LIN {X 0,Y 425.307,Z 310.007,A -85,B 0,C 180,E1 -9738.298,E2 -9738.298} C_VEL
LIN {X 0,Y 425.293,Z 310.002,A -85,B 0,C 180,E1 -9741.318,E2 -9741.318} C_VEL
LIN {X 0,Y 425.3,Z 309.999,A -85,B 0,C 180,E1 -9744.651,E2 -9744.651} C_VEL
LIN {X 0,Y 425.25,Z 310.01,A -85,B 0,C 180,E1 -9747.564,E2 -9747.564} C_VEL
LIN {X 0,Y 425.28,Z 310.001,A -85,B 0,C 180,E1 -9749.72,E2 -9749.72} C_VEL
LIN {X 0,Y 425.269,Z 310.007,A -85,B 0,C 180,E1 -9753.049,E2 -9753.049} C_VEL
LIN {X 0,Y 425.279,Z 310.005,A -85,B 0,C 180,E1 -9755.928,E2 -9755.928} C_VEL
LIN {X 0,Y 425.258,Z 310.007,A -85,B 0,C 180,E1 -9759.036,E2 -9759.036} C_VEL
LIN {X 0,Y 425.253,Z 310.008,A -85,B 0,C 180,E1 -9762.655,E2 -9762.655} C_VEL
LIN {X 0,Y 425.281,Z 310.005,A -85,B 0,C 180,E1 -9765.283,E2 -9765.283} C_VEL
LIN {X 0,Y 425.245,Z 310.016,A -85,B 0,C 180,E1 -9768.618,E2 -9768.618} C_VEL
LIN {X 0,Y 425.277,Z 310.011,A -85,B 0,C 180,E1 -9771.099,E2 -9771.099} C_VEL
LIN {X 0,Y 425.293,Z 310.007,A -85,B 0,C 180,E1 -9774.663,E2 -9774.663} C_VEL
LIN {X 0,Y 425.261,Z 310.012,A -85,B 0,C 180,E1 -9778.073,E2 -9778.073} C_VEL
LIN {X 0,Y 425.311,Z 310.005,A -85,B 0,C 180,E1 -9781.366,E2 -9781.366} C_VEL
LIN {X 0,Y 425.335,Z 310.116,A -85,B 0,C 180,E1 -9783.702,E2 -9783.702} C_VEL
LIN {X 0,Y 427.72,Z 322.373,A -85,B 0,C 180,E1 -9786.518,E2 -9786.518} C_VEL
LIN {X 0,Y 427.919,Z 326.115,A -85,B 0,C 180,E1 -9787.322,E2 -9787.322} C_VEL
LIN {X 0,Y 426.781,Z 342.849,A -85,B 0,C 180,E1 -9790.771,E2 -9790.771} C_VEL
LIN {X 0,Y 426.66,Z 345.828,A -85,B 0,C 180,E1 -9791.314,E2 -9791.314} C_VEL
LIN {X 0,Y 430.359,Z 367.602,A -85,B 0,C 180,E1 -9791.874,E2 -9791.874} C_VEL
LIN {X 0,Y 429.563,Z 451.981,A -85,B 0,C 180,E1 -9793.332,E2 -9793.332} C_VEL
LIN {X 0,Y 429.279,Z 461.728,A -85,B 0,C 180,E1 -9793.596,E2 -9793.596} C_VEL
LIN {X 0,Y 428.817,Z 472.261,A -85,B 0,C 180,E1 -9794.005,E2 -9794.005} C_VEL
LIN {X 0,Y 428.352,Z 482.441,A -85,B 0,C 180,E1 -9794.537,E2 -9794.537} C_VEL
LIN {X 0,Y 427.723,Z 493.013,A -85,B 0,C 180,E1 -9795.245,E2 -9795.245} C_VEL
LIN {X 0,Y 427.159,Z 502.459,A -85,B 0,C 180,E1 -9796.031,E2 -9796.031} C_VEL
LIN {X 0,Y 426.599,Z 511.193,A -85,B 0,C 180,E1 -9796.907,E2 -9796.907} C_VEL
LIN {X 0,Y 426.058,Z 519.156,A -85,B 0,C 180,E1 -9797.859,E2 -9797.859} C_VEL
LIN {X 0,Y 425.479,Z 527.402,A -85,B 0,C 180,E1 -9799.05,E2 -9799.05} C_VEL
LIN {X 0,Y 425.032,Z 534.27,A -85,B 0,C 180,E1 -9800.242,E2 -9800.242} C_VEL
LIN {X 0,Y 424.705,Z 540.013,A -85,B 0,C 180,E1 -9801.435,E2 -9801.435} C_VEL
LIN {X 0,Y 424.433,Z 545.574,A -85,B 0,C 180,E1 -9802.866,E2 -9802.866} C_VEL
LIN {X 0,Y 424.231,Z 549.948,A -85,B 0,C 180,E1 -9804.295,E2 -9804.295} C_VEL
LIN {X 0,Y 424.204,Z 552.264,A -85,B 0,C 180,E1 -9805.248,E2 -9805.248} C_VEL
LIN {X 0,Y 424.081,Z 555.578,A -85,B 0,C 180,E1 -9807.15,E2 -9807.15} C_VEL
LIN {X 0,Y 424.115,Z 556.545,A -85,B 0,C 180,E1 -9808.101,E2 -9808.101} C_VEL
LIN {X 0,Y 424.056,Z 557.441,A -85,B 0,C 180,E1 -9810,E2 -9810} C_VEL
LIN {X 0,Y 424.115,Z 556.603,A -85,B 0,C 180,E1 -9811.899,E2 -9811.899} C_VEL
LIN {X 0,Y 424.081,Z 555.632,A -85,B 0,C 180,E1 -9812.85,E2 -9812.85} C_VEL
LIN {X 0,Y 424.209,Z 552.407,A -85,B 0,C 180,E1 -9814.752,E2 -9814.752} C_VEL
LIN {X 0,Y 424.262,Z 548.344,A -85,B 0,C 180,E1 -9816.328,E2 -9816.328} C_VEL
LIN {X 0,Y 424.502,Z 544.103,A -85,B 0,C 180,E1 -9817.611,E2 -9817.611} C_VEL
LIN {X 0,Y 424.848,Z 538.126,A -85,B 0,C 180,E1 -9819.042,E2 -9819.042} C_VEL
LIN {X 0,Y 425.237,Z 532.082,A -85,B 0,C 180,E1 -9820.234,E2 -9820.234} C_VEL
LIN {X 0,Y 425.716,Z 524.793,A -85,B 0,C 180,E1 -9821.426,E2 -9821.426} C_VEL
LIN {X 0,Y 426.395,Z 515.929,A -85,B 0,C 180,E1 -9822.614,E2 -9822.614} C_VEL
LIN {X 0,Y 426.936,Z 506.91,A -85,B 0,C 180,E1 -9823.618,E2 -9823.618} C_VEL
LIN {X 0,Y 427.6,Z 497.037,A -85,B 0,C 180,E1 -9824.516,E2 -9824.516} C_VEL
LIN {X 0,Y 428.15,Z 487.502,A -85,B 0,C 180,E1 -9825.227,E2 -9825.227} C_VEL
LIN {X 0,Y 428.764,Z 477.643,A -85,B 0,C 180,E1 -9825.813,E2 -9825.813} C_VEL
LIN {X 0,Y 429.288,Z 465.878,A -85,B 0,C 180,E1 -9826.343,E2 -9826.343} C_VEL
LIN {X 0,Y 429.644,Z 455.964,A -85,B 0,C 180,E1 -9826.665,E2 -9826.665} C_VEL
LIN {X 0,Y 429.921,Z 439.713,A -85,B 0,C 180,E1 -9826.99,E2 -9826.99} C_VEL
LIN {X 0,Y 430.624,Z 368.061,A -85,B 0,C 180,E1 -9828.215,E2 -9828.215} C_VEL
LIN {X 0,Y 426.817,Z 345.669,A -85,B 0,C 180,E1 -9828.806,E2 -9828.806} C_VEL
LIN {X 0,Y 426.763,Z 344.428,A -85,B 0,C 180,E1 -9828.969,E2 -9828.969} C_VEL
LIN {X 0,Y 427.787,Z 327.218,A -85,B 0,C 180,E1 -9832.439,E2 -9832.439} C_VEL
LIN {X 0,Y 427.876,Z 323.444,A -85,B 0,C 180,E1 -9833.216,E2 -9833.216} C_VEL
LIN {X 0,Y 425.789,Z 312.361,A -85,B 0,C 180,E1 -9835.676,E2 -9835.676} C_VEL
LIN {X 0,Y 425.31,Z 310.053,A -85,B 0,C 180,E1 -9836.266,E2 -9836.266} C_VEL
LIN {X 0,Y 425.283,Z 310.01,A -85,B 0,C 180,E1 -9839.72,E2 -9839.72} C_VEL
LIN {X 0,Y 425.279,Z 310.009,A -85,B 0,C 180,E1 -9843.048,E2 -9843.048} C_VEL
LIN {X 0,Y 425.279,Z 310.009,A -85,B 0,C 180,E1 -9845.929,E2 -9845.929} C_VEL
LIN {X 0,Y 425.28,Z 310.008,A -85,B 0,C 180,E1 -9849.041,E2 -9849.041} C_VEL
LIN {X 0,Y 425.28,Z 310.007,A -85,B 0,C 180,E1 -9851.957,E2 -9851.957} C_VEL
LIN {X 0,Y 425.283,Z 310.011,A -85,B 0,C 180,E1 -9855.283,E2 -9855.283} C_VEL
LIN {X 0,Y 425.272,Z 310.004,A -85,B 0,C 180,E1 -9858.622,E2 -9858.622} C_VEL
LIN {X 0,Y 425.296,Z 310.005,A -85,B 0,C 180,E1 -9861.101,E2 -9861.101} C_VEL
LIN {X 0,Y 425.299,Z 310.001,A -85,B 0,C 180,E1 -9864.664,E2 -9864.664} C_VEL
LIN {X 0,Y 425.265,Z 310.012,A -85,B 0,C 180,E1 -9868.073,E2 -9868.073} C_VEL
LIN {X 0,Y 425.331,Z 309.999,A -85,B 0,C 180,E1 -9871.368,E2 -9871.368} C_VEL
LIN {X 0,Y 425.296,Z 310.009,A -85,B 0,C 180,E1 -9874.555,E2 -9874.555} C_VEL
LIN {X 0,Y 425.288,Z 310.004,A -85,B 0,C 180,E1 -9877.662,E2 -9877.662} C_VEL
LIN {X 0,Y 425.363,Z 309.997,A -85,B 0,C 180,E1 -9880.704,E2 -9880.704} C_VEL
LIN {X 0,Y 425.389,Z 309.996,A -85,B 0,C 180,E1 -9883.689,E2 -9883.689} C_VEL
LIN {X 0,Y 425.413,Z 309.991,A -85,B 0,C 180,E1 -9887.599,E2 -9887.599} C_VEL
LIN {X 0,Y 425.444,Z 309.981,A -85,B 0,C 180,E1 -9891.45,E2 -9891.45} C_VEL
LIN {X 0,Y 425.556,Z 309.974,A -85,B 0,C 180,E1 -9894.314,E2 -9894.314} C_VEL
LIN {X 0,Y 425.577,Z 309.972,A -85,B 0,C 180,E1 -9898.108,E2 -9898.108} C_VEL
LIN {X 0,Y 425.705,Z 309.952,A -85,B 0,C 180,E1 -9900,E2 -9900} C_VEL
LIN {X 0,Y 425.558,Z 309.978,A -85,B 0,C 180,E1 -9902.84,E2 -9902.84} C_VEL
LIN {X 0,Y 425.534,Z 309.977,A -85,B 0,C 180,E1 -9906.639,E2 -9906.639} C_VEL
LIN {X 0,Y 425.403,Z 309.995,A -85,B 0,C 180,E1 -9909.51,E2 -9909.51} C_VEL
LIN {X 0,Y 425.395,Z 309.989,A -85,B 0,C 180,E1 -9912.904,E2 -9912.904} C_VEL
LIN {X 0,Y 425.363,Z 309.995,A -85,B 0,C 180,E1 -9916.605,E2 -9916.605} C_VEL
LIN {X 0,Y 425.33,Z 310.001,A -85,B 0,C 180,E1 -9919.636,E2 -9919.636} C_VEL
LIN {X 0,Y 425.289,Z 310.01,A -85,B 0,C 180,E1 -9922.339,E2 -9922.339} C_VEL
LIN {X 0,Y 425.321,Z 310.006,A -85,B 0,C 180,E1 -9924.657,E2 -9924.657} C_VEL
LIN {X 0,Y 425.33,Z 309.992,A -85,B 0,C 180,E1 -9927.559,E2 -9927.559} C_VEL
LIN {X 0,Y 425.288,Z 310.006,A -85,B 0,C 180,E1 -9930.816,E2 -9930.816} C_VEL
LIN {X 0,Y 425.31,Z 310,A -85,B 0,C 180,E1 -9934.288,E2 -9934.288} C_VEL
LIN {X 0,Y 425.28,Z 310.01,A -85,B 0,C 180,E1 -9937.694,E2 -9937.694} C_VEL
LIN {X 0,Y 425.282,Z 310.011,A -85,B 0,C 180,E1 -9940.521,E2 -9940.521} C_VEL
LIN {X 0,Y 425.357,Z 310.083,A -85,B 0,C 180,E1 -9942.153,E2 -9942.153} C_VEL
LIN {X 0,Y 427.263,Z 319.771,A -85,B 0,C 180,E1 -9944.345,E2 -9944.345} C_VEL
LIN {X 0,Y 427.059,Z 329.794,A -85,B 0,C 180,E1 -9946.394,E2 -9946.394} C_VEL
LIN {X 0,Y 426.921,Z 334.032,A -85,B 0,C 180,E1 -9947.212,E2 -9947.212} C_VEL
LIN {X 0,Y 429.955,Z 350.192,A -85,B 0,C 180,E1 -9947.681,E2 -9947.681} C_VEL
LIN {X 0,Y 430.785,Z 356.193,A -85,B 0,C 180,E1 -9947.827,E2 -9947.827} C_VEL
LIN {X 0,Y 429.735,Z 440.182,A -85,B 0,C 180,E1 -9949.279,E2 -9949.279} C_VEL
LIN {X 0,Y 429.469,Z 450.36,A -85,B 0,C 180,E1 -9949.557,E2 -9949.557} C_VEL
LIN {X 0,Y 429.107,Z 461.311,A -85,B 0,C 180,E1 -9949.996,E2 -9949.996} C_VEL
LIN {X 0,Y 428.692,Z 470.759,A -85,B 0,C 180,E1 -9950.493,E2 -9950.493} C_VEL
LIN {X 0,Y 428.167,Z 480.146,A -85,B 0,C 180,E1 -9951.109,E2 -9951.109} C_VEL
LIN {X 0,Y 427.483,Z 490.943,A -85,B 0,C 180,E1 -9952.006,E2 -9952.006} C_VEL
LIN {X 0,Y 426.841,Z 499.891,A -85,B 0,C 180,E1 -9952.912,E2 -9952.912} C_VEL
LIN {X 0,Y 426.228,Z 508.549,A -85,B 0,C 180,E1 -9953.974,E2 -9953.974} C_VEL
LIN {X 0,Y 425.731,Z 515.487,A -85,B 0,C 180,E1 -9954.982,E2 -9954.982} C_VEL
LIN {X 0,Y 425.269,Z 521.992,A -85,B 0,C 180,E1 -9956.099,E2 -9956.099} C_VEL
LIN {X 0,Y 424.842,Z 528.755,A -85,B 0,C 180,E1 -9957.53,E2 -9957.53} C_VEL
LIN {X 0,Y 424.596,Z 532.91,A -85,B 0,C 180,E1 -9958.574,E2 -9958.574} C_VEL
LIN {X 0,Y 424.31,Z 537.98,A -85,B 0,C 180,E1 -9960.205,E2 -9960.205} C_VEL
LIN {X 0,Y 424.173,Z 540.902,A -85,B 0,C 180,E1 -9961.419,E2 -9961.419} C_VEL
LIN {X 0,Y 423.931,Z 544.018,A -85,B 0,C 180,E1 -9963.41,E2 -9963.41} C_VEL
LIN {X 0,Y 423.878,Z 545.06,A -85,B 0,C 180,E1 -9964.464,E2 -9964.464} C_VEL
LIN {X 0,Y 423.861,Z 545.528,A -85,B 0,C 180,E1 -9965.777,E2 -9965.777} C_VEL
LIN {X 0,Y 423.884,Z 545.029,A -85,B 0,C 180,E1 -9967.583,E2 -9967.583} C_VEL
LIN {X 0,Y 423.949,Z 543.998,A -85,B 0,C 180,E1 -9968.611,E2 -9968.611} C_VEL
LIN {X 0,Y 424.158,Z 540.764,A -85,B 0,C 180,E1 -9970.647,E2 -9970.647} C_VEL
LIN {X 0,Y 424.367,Z 536.989,A -85,B 0,C 180,E1 -9972.159,E2 -9972.159} C_VEL
LIN {X 0,Y 424.642,Z 531.745,A -85,B 0,C 180,E1 -9973.725,E2 -9973.725} C_VEL
LIN {X 0,Y 424.97,Z 525.693,A -85,B 0,C 180,E1 -9975.147,E2 -9975.147} C_VEL
LIN {X 0,Y 425.107,Z 523.362,A -85,B 0,C 180,E1 -9975.621,E2 -9975.621} C_VEL
LIN {X 0,Y 424.646,Z 520.061,A -85,B 0,C 180,E1 -9976.279,E2 -9976.279} C_VEL
LIN {X 0,Y 422.208,Z 514.295,A -85,B 0,C 180,E1 -9977.326,E2 -9977.326} C_VEL
LIN {X 0,Y 419.867,Z 507.939,A -85,B 0,C 180,E1 -9978.31,E2 -9978.31} C_VEL
LIN {X 0,Y 419.551,Z 503.63,A -85,B 0,C 180,E1 -9978.862,E2 -9978.862} C_VEL
LIN {X 0,Y 420.065,Z 495.684,A -85,B 0,C 180,E1 -9979.761,E2 -9979.761} C_VEL
LIN {X 0,Y 420.787,Z 486.221,A -85,B 0,C 180,E1 -9980.642,E2 -9980.642} C_VEL
LIN {X 0,Y 421.298,Z 476.851,A -85,B 0,C 180,E1 -9981.365,E2 -9981.365} C_VEL
LIN {X 0,Y 421.868,Z 465.719,A -85,B 0,C 180,E1 -9982.04,E2 -9982.04} C_VEL
LIN {X 0,Y 422.3,Z 455.141,A -85,B 0,C 180,E1 -9982.529,E2 -9982.529} C_VEL
LIN {X 0,Y 422.723,Z 443.786,A -85,B 0,C 180,E1 -9982.897,E2 -9982.897} C_VEL
LIN {X 0,Y 422.945,Z 427.148,A -85,B 0,C 180,E1 -9983.231,E2 -9983.231} C_VEL
LIN {X 0,Y 423.736,Z 355.549,A -85,B 0,C 180,E1 -9984.465,E2 -9984.465} C_VEL
LIN {X 0,Y 419.957,Z 335.166,A -85,B 0,C 180,E1 -9985.014,E2 -9985.014} C_VEL
LIN {X 0,Y 419.936,Z 333.83,A -85,B 0,C 180,E1 -9985.2,E2 -9985.2} C_VEL
LIN {X 0,Y 420.578,Z 323.19,A -85,B 0,C 180,E1 -9987.606,E2 -9987.606} C_VEL
LIN {X 0,Y 419.096,Z 313.301,A -85,B 0,C 180,E1 -9990,E2 -9990} C_VEL
LIN {X 0,Y 418.58,Z 310.893,A -85,B 0,C 180,E1 -9990.661,E2 -9990.661} C_VEL
LIN {X 0,Y 418.511,Z 310.857,A -85,B 0,C 180,E1 -9992.888,E2 -9992.888} C_VEL
LIN {X 0,Y 418.507,Z 310.849,A -85,B 0,C 180,E1 -9995.783,E2 -9995.783} C_VEL
LIN {X 0,Y 418.38,Z 310.864,A -85,B 0,C 180,E1 -9998.696,E2 -9998.696} C_VEL
LIN {X 0,Y 418.318,Z 310.873,A -85,B 0,C 180,E1 -10001.631,E2 -10001.631} C_VEL
LIN {X 0,Y 418.304,Z 310.874,A -85,B 0,C 180,E1 -10004.597,E2 -10004.597} C_VEL
LIN {X 0,Y 418.29,Z 310.88,A -85,B 0,C 180,E1 -10007.604,E2 -10007.604} C_VEL
LIN {X 0,Y 418.252,Z 310.886,A -85,B 0,C 180,E1 -10010.663,E2 -10010.663} C_VEL
LIN {X 0,Y 418.278,Z 310.873,A -85,B 0,C 180,E1 -10013.782,E2 -10013.782} C_VEL
LIN {X 0,Y 418.312,Z 310.874,A -85,B 0,C 180,E1 -10017.071,E2 -10017.071} C_VEL
LIN {X 0,Y 418.246,Z 310.881,A -85,B 0,C 180,E1 -10020.272,E2 -10020.272} C_VEL
LIN {X 0,Y 418.25,Z 310.876,A -85,B 0,C 180,E1 -10023.677,E2 -10023.677} C_VEL
LIN {X 0,Y 418.241,Z 310.883,A -85,B 0,C 180,E1 -10027.224,E2 -10027.224} C_VEL
LIN {X 0,Y 418.256,Z 310.884,A -85,B 0,C 180,E1 -10029.682,E2 -10029.682} C_VEL
LIN {X 0,Y 418.231,Z 310.878,A -85,B 0,C 180,E1 -10032.321,E2 -10032.321} C_VEL
LIN {X 0,Y 418.237,Z 310.884,A -85,B 0,C 180,E1 -10035.109,E2 -10035.109} C_VEL
LIN {X 0,Y 418.236,Z 310.88,A -85,B 0,C 180,E1 -10037.766,E2 -10037.766} C_VEL
LIN {X 0,Y 418.247,Z 310.875,A -85,B 0,C 180,E1 -10041.557,E2 -10041.557} C_VEL
LIN {X 0,Y 418.26,Z 310.884,A -85,B 0,C 180,E1 -10045.159,E2 -10045.159} C_VEL
LIN {X 0,Y 418.247,Z 310.883,A -85,B 0,C 180,E1 -10047.472,E2 -10047.472} C_VEL
LIN {X 0,Y 418.265,Z 310.858,A -85,B 0,C 180,E1 -10050.897,E2 -10050.897} C_VEL
LIN {X 0,Y 418.239,Z 310.884,A -85,B 0,C 180,E1 -10054.094,E2 -10054.094} C_VEL
LIN {X 0,Y 418.24,Z 310.881,A -85,B 0,C 180,E1 -10057.264,E2 -10057.264} C_VEL
LIN {X 0,Y 418.285,Z 310.869,A -85,B 0,C 180,E1 -10060.364,E2 -10060.364} C_VEL
LIN {X 0,Y 418.319,Z 310.864,A -85,B 0,C 180,E1 -10063.404,E2 -10063.404} C_VEL
LIN {X 0,Y 418.349,Z 310.871,A -85,B 0,C 180,E1 -10066.999,E2 -10066.999} C_VEL
LIN {X 0,Y 418.337,Z 310.864,A -85,B 0,C 180,E1 -10070.328,E2 -10070.328} C_VEL
LIN {X 0,Y 418.444,Z 310.84,A -85,B 0,C 180,E1 -10073.248,E2 -10073.248} C_VEL
LIN {X 0,Y 418.322,Z 310.857,A -85,B 0,C 180,E1 -10075.181,E2 -10075.181} C_VEL
LIN {X 0,Y 418.537,Z 310.847,A -85,B 0,C 180,E1 -10078.075,E2 -10078.075} C_VEL
LIN {X 0,Y 418.474,Z 310.851,A -85,B 0,C 180,E1 -10080.962,E2 -10080.962} C_VEL
LIN {X 0,Y 418.472,Z 310.844,A -85,B 0,C 180,E1 -10082.888,E2 -10082.888} C_VEL
LIN {X 0,Y 418.501,Z 310.835,A -85,B 0,C 180,E1 -10085.783,E2 -10085.783} C_VEL
LIN {X 0,Y 418.378,Z 310.864,A -85,B 0,C 180,E1 -10088.695,E2 -10088.695} C_VEL
LIN {X 0,Y 418.314,Z 310.875,A -85,B 0,C 180,E1 -10091.631,E2 -10091.631} C_VEL
LIN {X 0,Y 418.276,Z 310.862,A -85,B 0,C 180,E1 -10094.598,E2 -10094.598} C_VEL
LIN {X 0,Y 418.248,Z 310.879,A -85,B 0,C 180,E1 -10097.605,E2 -10097.605} C_VEL
LIN {X 0,Y 418.25,Z 310.882,A -85,B 0,C 180,E1 -10100.663,E2 -10100.663} C_VEL
LIN {X 0,Y 418.258,Z 310.869,A -85,B 0,C 180,E1 -10103.783,E2 -10103.783} C_VEL
LIN {X 0,Y 418.208,Z 310.891,A -85,B 0,C 180,E1 -10107.042,E2 -10107.042} C_VEL
LIN {X 0,Y 418.239,Z 310.878,A -85,B 0,C 180,E1 -10110.272,E2 -10110.272} C_VEL
LIN {X 0,Y 418.232,Z 310.888,A -85,B 0,C 180,E1 -10113.678,E2 -10113.678} C_VEL
LIN {X 0,Y 418.235,Z 310.882,A -85,B 0,C 180,E1 -10117.224,E2 -10117.224} C_VEL
LIN {X 0,Y 418.205,Z 310.886,A -85,B 0,C 180,E1 -10120.867,E2 -10120.867} C_VEL
LIN {X 0,Y 418.199,Z 310.887,A -85,B 0,C 180,E1 -10123.728,E2 -10123.728} C_VEL
LIN {X 0,Y 418.196,Z 310.892,A -85,B 0,C 180,E1 -10126.447,E2 -10126.447} C_VEL
LIN {X 0,Y 418.205,Z 310.89,A -85,B 0,C 180,E1 -10129.133,E2 -10129.133} C_VEL
LIN {X 0,Y 418.235,Z 310.888,A -85,B 0,C 180,E1 -10132.775,E2 -10132.775} C_VEL
LIN {X 0,Y 418.231,Z 310.879,A -85,B 0,C 180,E1 -10136.321,E2 -10136.321} C_VEL
LIN {X 0,Y 418.24,Z 310.887,A -85,B 0,C 180,E1 -10139.727,E2 -10139.727} C_VEL
LIN {X 0,Y 418.261,Z 310.883,A -85,B 0,C 180,E1 -10143.29,E2 -10143.29} C_VEL
LIN {X 0,Y 418.342,Z 311.312,A -85,B 0,C 180,E1 -10143.564,E2 -10143.564} C_VEL
LIN {X 0,Y 420.735,Z 323.434,A -85,B 0,C 180,E1 -10146.366,E2 -10146.366} C_VEL
LIN {X 0,Y 420.999,Z 326.557,A -85,B 0,C 180,E1 -10147.054,E2 -10147.054} C_VEL
LIN {X 0,Y 419.878,Z 342.711,A -85,B 0,C 180,E1 -10150.442,E2 -10150.442} C_VEL
LIN {X 0,Y 419.764,Z 345.804,A -85,B 0,C 180,E1 -10151.008,E2 -10151.008} C_VEL
LIN {X 0,Y 423.602,Z 368.605,A -85,B 0,C 180,E1 -10151.603,E2 -10151.603} C_VEL
LIN {X 0,Y 422.774,Z 451.411,A -85,B 0,C 180,E1 -10153.056,E2 -10153.056} C_VEL
LIN {X 0,Y 422.457,Z 461.325,A -85,B 0,C 180,E1 -10153.323,E2 -10153.323} C_VEL
LIN {X 0,Y 421.964,Z 471.943,A -85,B 0,C 180,E1 -10153.738,E2 -10153.738} C_VEL
LIN {X 0,Y 421.5,Z 482.178,A -85,B 0,C 180,E1 -10154.279,E2 -10154.279} C_VEL
LIN {X 0,Y 420.841,Z 492.786,A -85,B 0,C 180,E1 -10154.998,E2 -10154.998} C_VEL
LIN {X 0,Y 420.196,Z 502.896,A -85,B 0,C 180,E1 -10155.858,E2 -10155.858} C_VEL
LIN {X 0,Y 419.653,Z 511.008,A -85,B 0,C 180,E1 -10156.687,E2 -10156.687} C_VEL
LIN {X 0,Y 419.102,Z 518.987,A -85,B 0,C 180,E1 -10157.654,E2 -10157.654} C_VEL
LIN {X 0,Y 418.498,Z 527.245,A -85,B 0,C 180,E1 -10158.865,E2 -10158.865} C_VEL
LIN {X 0,Y 417.991,Z 534.123,A -85,B 0,C 180,E1 -10160.076,E2 -10160.076} C_VEL
LIN {X 0,Y 417.663,Z 539.876,A -85,B 0,C 180,E1 -10161.289,E2 -10161.289} C_VEL
LIN {X 0,Y 417.358,Z 545.445,A -85,B 0,C 180,E1 -10162.744,E2 -10162.744} C_VEL
LIN {X 0,Y 417.139,Z 549.827,A -85,B 0,C 180,E1 -10164.198,E2 -10164.198} C_VEL
LIN {X 0,Y 417.114,Z 552.143,A -85,B 0,C 180,E1 -10165.167,E2 -10165.167} C_VEL
LIN {X 0,Y 416.979,Z 555.47,A -85,B 0,C 180,E1 -10167.102,E2 -10167.102} C_VEL
LIN {X 0,Y 417.024,Z 556.438,A -85,B 0,C 180,E1 -10168.068,E2 -10168.068} C_VEL
LIN {X 0,Y 416.977,Z 557.342,A -85,B 0,C 180,E1 -10170,E2 -10170} C_VEL
LIN {X 0,Y 417.024,Z 556.512,A -85,B 0,C 180,E1 -10171.931,E2 -10171.931} C_VEL
LIN {X 0,Y 416.979,Z 555.539,A -85,B 0,C 180,E1 -10172.898,E2 -10172.898} C_VEL
LIN {X 0,Y 417.141,Z 552.324,A -85,B 0,C 180,E1 -10174.832,E2 -10174.832} C_VEL
LIN {X 0,Y 417.193,Z 548.597,A -85,B 0,C 180,E1 -10176.33,E2 -10176.33} C_VEL
LIN {X 0,Y 417.428,Z 544.029,A -85,B 0,C 180,E1 -10177.741,E2 -10177.741} C_VEL
LIN {X 0,Y 417.8,Z 538.056,A -85,B 0,C 180,E1 -10179.195,E2 -10179.195} C_VEL
LIN {X 0,Y 418.229,Z 532.023,A -85,B 0,C 180,E1 -10180.407,E2 -10180.407} C_VEL
LIN {X 0,Y 418.741,Z 524.747,A -85,B 0,C 180,E1 -10181.619,E2 -10181.619} C_VEL
LIN {X 0,Y 419.464,Z 515.899,A -85,B 0,C 180,E1 -10182.826,E2 -10182.826} C_VEL
LIN {X 0,Y 420.023,Z 506.902,A -85,B 0,C 180,E1 -10183.846,E2 -10183.846} C_VEL
LIN {X 0,Y 420.702,Z 497.057,A -85,B 0,C 180,E1 -10184.759,E2 -10184.759} C_VEL
LIN {X 0,Y 421.295,Z 487.553,A -85,B 0,C 180,E1 -10185.48,E2 -10185.48} C_VEL
LIN {X 0,Y 421.949,Z 477.738,A -85,B 0,C 180,E1 -10186.076,E2 -10186.076} C_VEL
LIN {X 0,Y 422.496,Z 466.046,A -85,B 0,C 180,E1 -10186.613,E2 -10186.613} C_VEL
LIN {X 0,Y 422.924,Z 455,A -85,B 0,C 180,E1 -10186.969,E2 -10186.969} C_VEL
LIN {X 0,Y 423.161,Z 440.198,A -85,B 0,C 180,E1 -10187.27,E2 -10187.27} C_VEL
LIN {X 0,Y 423.844,Z 368.772,A -85,B 0,C 180,E1 -10188.514,E2 -10188.514} C_VEL
LIN {X 0,Y 419.854,Z 345.338,A -85,B 0,C 180,E1 -10189.158,E2 -10189.158} C_VEL
LIN {X 0,Y 420.105,Z 340.764,A -85,B 0,C 180,E1 -10190.024,E2 -10190.024} C_VEL
LIN {X 0,Y 421.004,Z 326.551,A -85,B 0,C 180,E1 -10192.949,E2 -10192.949} C_VEL
LIN {X 0,Y 420.3,Z 320.926,A -85,B 0,C 180,E1 -10194.184,E2 -10194.184} C_VEL
LIN {X 0,Y 418.283,Z 310.988,A -85,B 0,C 180,E1 -10196.507,E2 -10196.507} C_VEL
LIN {X 0,Y 418.258,Z 310.886,A -85,B 0,C 180,E1 -10199.162,E2 -10199.162} C_VEL
LIN {X 0,Y 418.255,Z 310.886,A -85,B 0,C 180,E1 -10202.844,E2 -10202.844} C_VEL
LIN {X 0,Y 418.242,Z 310.886,A -85,B 0,C 180,E1 -10206.238,E2 -10206.238} C_VEL
LIN {X 0,Y 418.242,Z 310.879,A -85,B 0,C 180,E1 -10209.683,E2 -10209.683} C_VEL
LIN {X 0,Y 418.222,Z 310.887,A -85,B 0,C 180,E1 -10212.32,E2 -10212.32} C_VEL
LIN {X 0,Y 418.234,Z 310.89,A -85,B 0,C 180,E1 -10215.109,E2 -10215.109} C_VEL
LIN {X 0,Y 418.239,Z 310.885,A -85,B 0,C 180,E1 -10217.767,E2 -10217.767} C_VEL
LIN {X 0,Y 418.244,Z 310.882,A -85,B 0,C 180,E1 -10220.621,E2 -10220.621} C_VEL
LIN {X 0,Y 418.243,Z 310.886,A -85,B 0,C 180,E1 -10223.976,E2 -10223.976} C_VEL
LIN {X 0,Y 418.257,Z 310.881,A -85,B 0,C 180,E1 -10227.156,E2 -10227.156} C_VEL
LIN {X 0,Y 418.268,Z 310.881,A -85,B 0,C 180,E1 -10230.896,E2 -10230.896} C_VEL
LIN {X 0,Y 418.271,Z 310.879,A -85,B 0,C 180,E1 -10234.096,E2 -10234.096} C_VEL
LIN {X 0,Y 418.238,Z 310.884,A -85,B 0,C 180,E1 -10237.264,E2 -10237.264} C_VEL
LIN {X 0,Y 418.284,Z 310.877,A -85,B 0,C 180,E1 -10240.365,E2 -10240.365} C_VEL
LIN {X 0,Y 418.318,Z 310.879,A -85,B 0,C 180,E1 -10243.405,E2 -10243.405} C_VEL
LIN {X 0,Y 418.347,Z 310.865,A -85,B 0,C 180,E1 -10246.999,E2 -10246.999} C_VEL
LIN {X 0,Y 418.343,Z 310.866,A -85,B 0,C 180,E1 -10250.329,E2 -10250.329} C_VEL
LIN {X 0,Y 418.495,Z 310.851,A -85,B 0,C 180,E1 -10253.249,E2 -10253.249} C_VEL
LIN {X 0,Y 418.342,Z 310.866,A -85,B 0,C 180,E1 -10255.182,E2 -10255.182} C_VEL
LIN {X 0,Y 418.546,Z 310.848,A -85,B 0,C 180,E1 -10258.076,E2 -10258.076} C_VEL
LIN {X 0,Y 418.675,Z 310.828,A -85,B 0,C 180,E1 -10260,E2 -10260} C_VEL
LIN {X 0,Y 418.511,Z 310.855,A -85,B 0,C 180,E1 -10262.888,E2 -10262.888} C_VEL
LIN {X 0,Y 418.497,Z 310.854,A -85,B 0,C 180,E1 -10266.751,E2 -10266.751} C_VEL
LIN {X 0,Y 418.343,Z 310.873,A -85,B 0,C 180,E1 -10269.672,E2 -10269.672} C_VEL
LIN {X 0,Y 418.348,Z 310.868,A -85,B 0,C 180,E1 -10273.001,E2 -10273.001} C_VEL
LIN {X 0,Y 418.315,Z 310.873,A -85,B 0,C 180,E1 -10276.736,E2 -10276.736} C_VEL
LIN {X 0,Y 418.272,Z 310.881,A -85,B 0,C 180,E1 -10279.791,E2 -10279.791} C_VEL
LIN {X 0,Y 418.233,Z 310.887,A -85,B 0,C 180,E1 -10282.737,E2 -10282.737} C_VEL
LIN {X 0,Y 418.24,Z 310.886,A -85,B 0,C 180,E1 -10285.906,E2 -10285.906} C_VEL
LIN {X 0,Y 418.265,Z 310.884,A -85,B 0,C 180,E1 -10289.162,E2 -10289.162} C_VEL
LIN {X 0,Y 418.258,Z 310.888,A -85,B 0,C 180,E1 -10292.844,E2 -10292.844} C_VEL
LIN {X 0,Y 418.245,Z 310.883,A -85,B 0,C 180,E1 -10296.238,E2 -10296.238} C_VEL
LIN {X 0,Y 418.252,Z 310.886,A -85,B 0,C 180,E1 -10299.682,E2 -10299.682} C_VEL
LIN {X 0,Y 418.295,Z 311.004,A -85,B 0,C 180,E1 -10301.902,E2 -10301.902} C_VEL
LIN {X 0,Y 420.323,Z 321.063,A -85,B 0,C 180,E1 -10304.21,E2 -10304.21} C_VEL
LIN {X 0,Y 420.155,Z 330.393,A -85,B 0,C 180,E1 -10306.151,E2 -10306.151} C_VEL
LIN {X 0,Y 420.037,Z 334.284,A -85,B 0,C 180,E1 -10306.892,E2 -10306.892} C_VEL
LIN {X 0,Y 424.041,Z 355.674,A -85,B 0,C 180,E1 -10307.503,E2 -10307.503} C_VEL
LIN {X 0,Y 422.984,Z 440.635,A -85,B 0,C 180,E1 -10309.001,E2 -10309.001} C_VEL
LIN {X 0,Y 422.699,Z 450.667,A -85,B 0,C 180,E1 -10309.283,E2 -10309.283} C_VEL
LIN {X 0,Y 422.345,Z 460.716,A -85,B 0,C 180,E1 -10309.686,E2 -10309.686} C_VEL
LIN {X 0,Y 421.874,Z 470.893,A -85,B 0,C 180,E1 -10310.227,E2 -10310.227} C_VEL
LIN {X 0,Y 421.215,Z 481.625,A -85,B 0,C 180,E1 -10310.961,E2 -10310.961} C_VEL
LIN {X 0,Y 420.56,Z 491.518,A -85,B 0,C 180,E1 -10311.807,E2 -10311.807} C_VEL
LIN {X 0,Y 419.945,Z 499.733,A -85,B 0,C 180,E1 -10312.651,E2 -10312.651} C_VEL
LIN {X 0,Y 419.405,Z 507.138,A -85,B 0,C 180,E1 -10313.547,E2 -10313.547} C_VEL
LIN {X 0,Y 418.702,Z 516.299,A -85,B 0,C 180,E1 -10314.908,E2 -10314.908} C_VEL
LIN {X 0,Y 418.219,Z 522.612,A -85,B 0,C 180,E1 -10316.03,E2 -10316.03} C_VEL
LIN {X 0,Y 417.785,Z 529.066,A -85,B 0,C 180,E1 -10317.432,E2 -10317.432} C_VEL
LIN {X 0,Y 417.514,Z 533.372,A -85,B 0,C 180,E1 -10318.545,E2 -10318.545} C_VEL
LIN {X 0,Y 417.229,Z 538.331,A -85,B 0,C 180,E1 -10320.204,E2 -10320.204} C_VEL
LIN {X 0,Y 417.026,Z 541.901,A -85,B 0,C 180,E1 -10321.844,E2 -10321.844} C_VEL
LIN {X 0,Y 416.837,Z 544.091,A -85,B 0,C 180,E1 -10323.329,E2 -10323.329} C_VEL
LIN {X 0,Y 416.76,Z 545.399,A -85,B 0,C 180,E1 -10325.065,E2 -10325.065} C_VEL
LIN {X 0,Y 416.764,Z 545.663,A -85,B 0,C 180,E1 -10326.127,E2 -10326.127} C_VEL
LIN {X 0,Y 416.81,Z 544.713,A -85,B 0,C 180,E1 -10328.03,E2 -10328.03} C_VEL
LIN {X 0,Y 416.909,Z 543.364,A -85,B 0,C 180,E1 -10329.268,E2 -10329.268} C_VEL
LIN {X 0,Y 417.088,Z 540.97,A -85,B 0,C 180,E1 -10330.667,E2 -10330.667} C_VEL
LIN {X 0,Y 417.308,Z 536.774,A -85,B 0,C 180,E1 -10332.354,E2 -10332.354} C_VEL
LIN {X 0,Y 417.542,Z 532.726,A -85,B 0,C 180,E1 -10333.621,E2 -10333.621} C_VEL
LIN {X 0,Y 417.899,Z 526.528,A -85,B 0,C 180,E1 -10335.14,E2 -10335.14} C_VEL
LIN {X 0,Y 418.349,Z 520.24,A -85,B 0,C 180,E1 -10336.397,E2 -10336.397} C_VEL
LIN {X 0,Y 418.871,Z 512.645,A -85,B 0,C 180,E1 -10337.648,E2 -10337.648} C_VEL
LIN {X 0,Y 419.551,Z 503.63,A -85,B 0,C 180,E1 -10338.862,E2 -10338.862} C_VEL
LIN {X 0,Y 419.099,Z 500.724,A -85,B 0,C 180,E1 -10339.228,E2 -10339.228} C_VEL
LIN {X 0,Y 416.592,Z 496.166,A -85,B 0,C 180,E1 -10339.83,E2 -10339.83} C_VEL
LIN {X 0,Y 414.133,Z 491.448,A -85,B 0,C 180,E1 -10340.403,E2 -10340.403} C_VEL
LIN {X 0,Y 413.749,Z 488.213,A -85,B 0,C 180,E1 -10340.718,E2 -10340.718} C_VEL
LIN {X 0,Y 414.408,Z 477.279,A -85,B 0,C 180,E1 -10341.589,E2 -10341.589} C_VEL
LIN {X 0,Y 415.003,Z 466.238,A -85,B 0,C 180,E1 -10342.275,E2 -10342.275} C_VEL
LIN {X 0,Y 415.491,Z 454.954,A -85,B 0,C 180,E1 -10342.803,E2 -10342.803} C_VEL
LIN {X 0,Y 415.877,Z 444.808,A -85,B 0,C 180,E1 -10343.145,E2 -10343.145} C_VEL
LIN {X 0,Y 416.164,Z 426.647,A -85,B 0,C 180,E1 -10343.516,E2 -10343.516} C_VEL
LIN {X 0,Y 416.91,Z 355.793,A -85,B 0,C 180,E1 -10344.761,E2 -10344.761} C_VEL
LIN {X 0,Y 413.051,Z 335.189,A -85,B 0,C 180,E1 -10345.334,E2 -10345.334} C_VEL
LIN {X 0,Y 413.016,Z 334.089,A -85,B 0,C 180,E1 -10345.486,E2 -10345.486} C_VEL
LIN {X 0,Y 413.582,Z 323.981,A -85,B 0,C 180,E1 -10347.809,E2 -10347.809} C_VEL
LIN {X 0,Y 411.823,Z 313.159,A -85,B 0,C 180,E1 -10350.489,E2 -10350.489} C_VEL
LIN {X 0,Y 411.474,Z 311.76,A -85,B 0,C 180,E1 -10350.918,E2 -10350.918} C_VEL
LIN {X 0,Y 411.466,Z 311.734,A -85,B 0,C 180,E1 -10352.937,E2 -10352.937} C_VEL
LIN {X 0,Y 411.468,Z 311.725,A -85,B 0,C 180,E1 -10355.882,E2 -10355.882} C_VEL
LIN {X 0,Y 411.321,Z 311.744,A -85,B 0,C 180,E1 -10358.846,E2 -10358.846} C_VEL
LIN {X 0,Y 411.286,Z 311.748,A -85,B 0,C 180,E1 -10361.833,E2 -10361.833} C_VEL
LIN {X 0,Y 411.261,Z 311.751,A -85,B 0,C 180,E1 -10364.853,E2 -10364.853} C_VEL
LIN {X 0,Y 411.255,Z 311.759,A -85,B 0,C 180,E1 -10367.915,E2 -10367.915} C_VEL
LIN {X 0,Y 411.198,Z 311.761,A -85,B 0,C 180,E1 -10371.034,E2 -10371.034} C_VEL
LIN {X 0,Y 411.222,Z 311.755,A -85,B 0,C 180,E1 -10374.216,E2 -10374.216} C_VEL
LIN {X 0,Y 411.261,Z 311.747,A -85,B 0,C 180,E1 -10377.478,E2 -10377.478} C_VEL
LIN {X 0,Y 411.191,Z 311.763,A -85,B 0,C 180,E1 -10380.848,E2 -10380.848} C_VEL
LIN {X 0,Y 411.207,Z 311.749,A -85,B 0,C 180,E1 -10384.334,E2 -10384.334} C_VEL
LIN {X 0,Y 411.197,Z 311.766,A -85,B 0,C 180,E1 -10387.974,E2 -10387.974} C_VEL
LIN {X 0,Y 411.185,Z 311.754,A -85,B 0,C 180,E1 -10390.504,E2 -10390.504} C_VEL
LIN {X 0,Y 411.174,Z 311.757,A -85,B 0,C 180,E1 -10393.134,E2 -10393.134} C_VEL
LIN {X 0,Y 411.169,Z 311.764,A -85,B 0,C 180,E1 -10395.881,E2 -10395.881} C_VEL
LIN {X 0,Y 411.16,Z 311.76,A -85,B 0,C 180,E1 -10398.773,E2 -10398.773} C_VEL
LIN {X 0,Y 411.192,Z 311.751,A -85,B 0,C 180,E1 -10402.026,E2 -10402.026} C_VEL
LIN {X 0,Y 411.207,Z 311.762,A -85,B 0,C 180,E1 -10405.666,E2 -10405.666} C_VEL
LIN {X 0,Y 411.191,Z 311.753,A -85,B 0,C 180,E1 -10409.152,E2 -10409.152} C_VEL
LIN {X 0,Y 411.19,Z 311.755,A -85,B 0,C 180,E1 -10412.517,E2 -10412.517} C_VEL
LIN {X 0,Y 411.22,Z 311.758,A -85,B 0,C 180,E1 -10415.784,E2 -10415.784} C_VEL
LIN {X 0,Y 411.199,Z 311.753,A -85,B 0,C 180,E1 -10418.966,E2 -10418.966} C_VEL
LIN {X 0,Y 411.247,Z 311.729,A -85,B 0,C 180,E1 -10422.085,E2 -10422.085} C_VEL
LIN {X 0,Y 411.26,Z 311.751,A -85,B 0,C 180,E1 -10425.147,E2 -10425.147} C_VEL
LIN {X 0,Y 411.284,Z 311.748,A -85,B 0,C 180,E1 -10428.167,E2 -10428.167} C_VEL
LIN {X 0,Y 411.318,Z 311.74,A -85,B 0,C 180,E1 -10431.154,E2 -10431.154} C_VEL
LIN {X 0,Y 411.432,Z 311.714,A -85,B 0,C 180,E1 -10434.117,E2 -10434.117} C_VEL
LIN {X 0,Y 411.505,Z 311.722,A -85,B 0,C 180,E1 -10438.042,E2 -10438.042} C_VEL
LIN {X 0,Y 411.438,Z 311.727,A -85,B 0,C 180,E1 -10440.979,E2 -10440.979} C_VEL
LIN {X 0,Y 411.43,Z 311.72,A -85,B 0,C 180,E1 -10442.937,E2 -10442.937} C_VEL
LIN {X 0,Y 411.434,Z 311.722,A -85,B 0,C 180,E1 -10446.867,E2 -10446.867} C_VEL
LIN {X 0,Y 411.289,Z 311.75,A -85,B 0,C 180,E1 -10449.839,E2 -10449.839} C_VEL
LIN {X 0,Y 411.307,Z 311.745,A -85,B 0,C 180,E1 -10453.104,E2 -10453.104} C_VEL
LIN {X 0,Y 411.209,Z 311.751,A -85,B 0,C 180,E1 -10456.89,E2 -10456.89} C_VEL
LIN {X 0,Y 411.232,Z 311.762,A -85,B 0,C 180,E1 -10459.986,E2 -10459.986} C_VEL
LIN {X 0,Y 411.189,Z 311.749,A -85,B 0,C 180,E1 -10463.148,E2 -10463.148} C_VEL
LIN {X 0,Y 411.175,Z 311.762,A -85,B 0,C 180,E1 -10466.385,E2 -10466.385} C_VEL
LIN {X 0,Y 411.196,Z 311.756,A -85,B 0,C 180,E1 -10469.713,E2 -10469.713} C_VEL
LIN {X 0,Y 411.204,Z 311.76,A -85,B 0,C 180,E1 -10473.156,E2 -10473.156} C_VEL
LIN {X 0,Y 411.19,Z 311.756,A -85,B 0,C 180,E1 -10476.552,E2 -10476.552} C_VEL
LIN {X 0,Y 411.167,Z 311.769,A -85,B 0,C 180,E1 -10479.72,E2 -10479.72} C_VEL
LIN {X 0,Y 411.159,Z 311.762,A -85,B 0,C 180,E1 -10483.135,E2 -10483.135} C_VEL
LIN {X 0,Y 411.161,Z 311.766,A -85,B 0,C 180,E1 -10485.882,E2 -10485.882} C_VEL
LIN {X 0,Y 411.156,Z 311.766,A -85,B 0,C 180,E1 -10489.493,E2 -10489.493} C_VEL
LIN {X 0,Y 411.183,Z 311.762,A -85,B 0,C 180,E1 -10492.025,E2 -10492.025} C_VEL
LIN {X 0,Y 411.201,Z 311.766,A -85,B 0,C 180,E1 -10495.123,E2 -10495.123} C_VEL
LIN {X 0,Y 411.162,Z 311.769,A -85,B 0,C 180,E1 -10498.002,E2 -10498.002} C_VEL
LIN {X 0,Y 411.192,Z 311.763,A -85,B 0,C 180,E1 -10501.408,E2 -10501.408} C_VEL
LIN {X 0,Y 411.245,Z 311.918,A -85,B 0,C 180,E1 -10503.22,E2 -10503.22} C_VEL
LIN {X 0,Y 413.496,Z 323.273,A -85,B 0,C 180,E1 -10505.926,E2 -10505.926} C_VEL
LIN {X 0,Y 414.005,Z 328.116,A -85,B 0,C 180,E1 -10507.018,E2 -10507.018} C_VEL
LIN {X 0,Y 412.903,Z 343.76,A -85,B 0,C 180,E1 -10510.357,E2 -10510.357} C_VEL
LIN {X 0,Y 412.811,Z 345.538,A -85,B 0,C 180,E1 -10510.676,E2 -10510.676} C_VEL
LIN {X 0,Y 416.889,Z 370.008,A -85,B 0,C 180,E1 -10511.335,E2 -10511.335} C_VEL
LIN {X 0,Y 415.964,Z 450.706,A -85,B 0,C 180,E1 -10512.77,E2 -10512.77} C_VEL
LIN {X 0,Y 415.625,Z 461.666,A -85,B 0,C 180,E1 -10513.072,E2 -10513.072} C_VEL
LIN {X 0,Y 415.128,Z 471.556,A -85,B 0,C 180,E1 -10513.463,E2 -10513.463} C_VEL
LIN {X 0,Y 414.656,Z 481.856,A -85,B 0,C 180,E1 -10514.013,E2 -10514.013} C_VEL
LIN {X 0,Y 413.961,Z 492.508,A -85,B 0,C 180,E1 -10514.743,E2 -10514.743} C_VEL
LIN {X 0,Y 413.323,Z 502.321,A -85,B 0,C 180,E1 -10515.584,E2 -10515.584} C_VEL
LIN {X 0,Y 412.714,Z 510.795,A -85,B 0,C 180,E1 -10516.459,E2 -10516.459} C_VEL
LIN {X 0,Y 412.153,Z 518.797,A -85,B 0,C 180,E1 -10517.443,E2 -10517.443} C_VEL
LIN {X 0,Y 411.509,Z 527.074,A -85,B 0,C 180,E1 -10518.673,E2 -10518.673} C_VEL
LIN {X 0,Y 410.975,Z 533.967,A -85,B 0,C 180,E1 -10519.905,E2 -10519.905} C_VEL
LIN {X 0,Y 410.603,Z 539.733,A -85,B 0,C 180,E1 -10521.138,E2 -10521.138} C_VEL
LIN {X 0,Y 410.285,Z 545.314,A -85,B 0,C 180,E1 -10522.619,E2 -10522.619} C_VEL
LIN {X 0,Y 410.064,Z 549.705,A -85,B 0,C 180,E1 -10524.098,E2 -10524.098} C_VEL
LIN {X 0,Y 410.029,Z 552.022,A -85,B 0,C 180,E1 -10525.084,E2 -10525.084} C_VEL
LIN {X 0,Y 409.878,Z 555.362,A -85,B 0,C 180,E1 -10527.051,E2 -10527.051} C_VEL
LIN {X 0,Y 409.912,Z 556.935,A -85,B 0,C 180,E1 -10529.018,E2 -10529.018} C_VEL
LIN {X 0,Y 409.901,Z 557.242,A -85,B 0,C 180,E1 -10530,E2 -10530} C_VEL
LIN {X 0,Y 409.92,Z 556.42,A -85,B 0,C 180,E1 -10531.965,E2 -10531.965} C_VEL
LIN {X 0,Y 409.878,Z 555.447,A -85,B 0,C 180,E1 -10532.948,E2 -10532.948} C_VEL
LIN {X 0,Y 410.052,Z 552.244,A -85,B 0,C 180,E1 -10534.916,E2 -10534.916} C_VEL
LIN {X 0,Y 410.115,Z 548.88,A -85,B 0,C 180,E1 -10536.322,E2 -10536.322} C_VEL
LIN {X 0,Y 410.374,Z 543.967,A -85,B 0,C 180,E1 -10537.875,E2 -10537.875} C_VEL
LIN {X 0,Y 410.749,Z 538.006,A -85,B 0,C 180,E1 -10539.355,E2 -10539.355} C_VEL
LIN {X 0,Y 411.222,Z 531.982,A -85,B 0,C 180,E1 -10540.587,E2 -10540.587} C_VEL
LIN {X 0,Y 411.779,Z 524.717,A -85,B 0,C 180,E1 -10541.818,E2 -10541.818} C_VEL
LIN {X 0,Y 412.536,Z 515.882,A -85,B 0,C 180,E1 -10543.046,E2 -10543.046} C_VEL
LIN {X 0,Y 413.101,Z 507.186,A -85,B 0,C 180,E1 -10544.054,E2 -10544.054} C_VEL
LIN {X 0,Y 413.829,Z 497.078,A -85,B 0,C 180,E1 -10545.01,E2 -10545.01} C_VEL
LIN {X 0,Y 414.478,Z 487.603,A -85,B 0,C 180,E1 -10545.742,E2 -10545.742} C_VEL
LIN {X 0,Y 415.21,Z 476.625,A -85,B 0,C 180,E1 -10546.407,E2 -10546.407} C_VEL
LIN {X 0,Y 415.72,Z 466.215,A -85,B 0,C 180,E1 -10546.892,E2 -10546.892} C_VEL
LIN {X 0,Y 416.159,Z 455.322,A -85,B 0,C 180,E1 -10547.253,E2 -10547.253} C_VEL
LIN {X 0,Y 416.415,Z 440.683,A -85,B 0,C 180,E1 -10547.559,E2 -10547.559} C_VEL
LIN {X 0,Y 417.166,Z 369.814,A -85,B 0,C 180,E1 -10548.812,E2 -10548.812} C_VEL
LIN {X 0,Y 412.989,Z 345.398,A -85,B 0,C 180,E1 -10549.492,E2 -10549.492} C_VEL
LIN {X 0,Y 413.061,Z 343.013,A -85,B 0,C 180,E1 -10549.894,E2 -10549.894} C_VEL
LIN {X 0,Y 414.045,Z 328.267,A -85,B 0,C 180,E1 -10552.979,E2 -10552.979} C_VEL
LIN {X 0,Y 413.57,Z 323.345,A -85,B 0,C 180,E1 -10554.069,E2 -10554.069} C_VEL
LIN {X 0,Y 411.238,Z 311.895,A -85,B 0,C 180,E1 -10556.78,E2 -10556.78} C_VEL
LIN {X 0,Y 411.195,Z 311.765,A -85,B 0,C 180,E1 -10559.713,E2 -10559.713} C_VEL
LIN {X 0,Y 411.204,Z 311.762,A -85,B 0,C 180,E1 -10563.156,E2 -10563.156} C_VEL
LIN {X 0,Y 411.19,Z 311.762,A -85,B 0,C 180,E1 -10566.553,E2 -10566.553} C_VEL
LIN {X 0,Y 411.207,Z 311.755,A -85,B 0,C 180,E1 -10569.727,E2 -10569.727} C_VEL
LIN {X 0,Y 411.169,Z 311.769,A -85,B 0,C 180,E1 -10573.134,E2 -10573.134} C_VEL
LIN {X 0,Y 411.166,Z 311.766,A -85,B 0,C 180,E1 -10575.881,E2 -10575.881} C_VEL
LIN {X 0,Y 411.162,Z 311.762,A -85,B 0,C 180,E1 -10578.772,E2 -10578.772} C_VEL
LIN {X 0,Y 411.191,Z 311.765,A -85,B 0,C 180,E1 -10582.026,E2 -10582.026} C_VEL
LIN {X 0,Y 411.205,Z 311.758,A -85,B 0,C 180,E1 -10585.667,E2 -10585.667} C_VEL
LIN {X 0,Y 411.189,Z 311.76,A -85,B 0,C 180,E1 -10589.153,E2 -10589.153} C_VEL
LIN {X 0,Y 411.259,Z 311.753,A -85,B 0,C 180,E1 -10592.523,E2 -10592.523} C_VEL
LIN {X 0,Y 411.227,Z 311.755,A -85,B 0,C 180,E1 -10595.785,E2 -10595.785} C_VEL
LIN {X 0,Y 411.197,Z 311.766,A -85,B 0,C 180,E1 -10598.966,E2 -10598.966} C_VEL
LIN {X 0,Y 411.253,Z 311.75,A -85,B 0,C 180,E1 -10602.085,E2 -10602.085} C_VEL
LIN {X 0,Y 411.262,Z 311.756,A -85,B 0,C 180,E1 -10605.148,E2 -10605.148} C_VEL
LIN {X 0,Y 411.285,Z 311.752,A -85,B 0,C 180,E1 -10608.168,E2 -10608.168} C_VEL
LIN {X 0,Y 411.483,Z 311.727,A -85,B 0,C 180,E1 -10612.147,E2 -10612.147} C_VEL
LIN {X 0,Y 411.477,Z 311.731,A -85,B 0,C 180,E1 -10614.118,E2 -10614.118} C_VEL
LIN {X 0,Y 411.515,Z 311.723,A -85,B 0,C 180,E1 -10618.043,E2 -10618.043} C_VEL
LIN {X 0,Y 411.644,Z 311.704,A -85,B 0,C 180,E1 -10620,E2 -10620} C_VEL
LIN {X 0,Y 411.467,Z 311.731,A -85,B 0,C 180,E1 -10622.937,E2 -10622.937} C_VEL
LIN {X 0,Y 411.463,Z 311.732,A -85,B 0,C 180,E1 -10626.867,E2 -10626.867} C_VEL
LIN {X 0,Y 411.295,Z 311.75,A -85,B 0,C 180,E1 -10629.839,E2 -10629.839} C_VEL
LIN {X 0,Y 411.307,Z 311.745,A -85,B 0,C 180,E1 -10633.104,E2 -10633.104} C_VEL
LIN {X 0,Y 411.259,Z 311.752,A -85,B 0,C 180,E1 -10636.889,E2 -10636.889} C_VEL
LIN {X 0,Y 411.232,Z 311.76,A -85,B 0,C 180,E1 -10639.987,E2 -10639.987} C_VEL
LIN {X 0,Y 411.197,Z 311.762,A -85,B 0,C 180,E1 -10643.148,E2 -10643.148} C_VEL
LIN {X 0,Y 411.205,Z 311.762,A -85,B 0,C 180,E1 -10646.383,E2 -10646.383} C_VEL
LIN {X 0,Y 411.201,Z 311.762,A -85,B 0,C 180,E1 -10649.713,E2 -10649.713} C_VEL
LIN {X 0,Y 411.207,Z 311.763,A -85,B 0,C 180,E1 -10653.156,E2 -10653.156} C_VEL
LIN {X 0,Y 411.193,Z 311.761,A -85,B 0,C 180,E1 -10656.553,E2 -10656.553} C_VEL
LIN {X 0,Y 411.216,Z 311.762,A -85,B 0,C 180,E1 -10659.728,E2 -10659.728} C_VEL
LIN {X 0,Y 411.24,Z 311.887,A -85,B 0,C 180,E1 -10661.618,E2 -10661.618} C_VEL
LIN {X 0,Y 413.454,Z 322.859,A -85,B 0,C 180,E1 -10664.181,E2 -10664.181} C_VEL
LIN {X 0,Y 413.139,Z 333.247,A -85,B 0,C 180,E1 -10666.358,E2 -10666.358} C_VEL
LIN {X 0,Y 413.175,Z 334.58,A -85,B 0,C 180,E1 -10666.556,E2 -10666.556} C_VEL
LIN {X 0,Y 417.302,Z 356.299,A -85,B 0,C 180,E1 -10667.189,E2 -10667.189} C_VEL
LIN {X 0,Y 416.221,Z 441.059,A -85,B 0,C 180,E1 -10668.713,E2 -10668.713} C_VEL
LIN {X 0,Y 415.922,Z 450.812,A -85,B 0,C 180,E1 -10668.992,E2 -10668.992} C_VEL
LIN {X 0,Y 415.559,Z 460.997,A -85,B 0,C 180,E1 -10669.41,E2 -10669.41} C_VEL
LIN {X 0,Y 415.056,Z 471.016,A -85,B 0,C 180,E1 -10669.951,E2 -10669.951} C_VEL
LIN {X 0,Y 414.419,Z 481.367,A -85,B 0,C 180,E1 -10670.667,E2 -10670.667} C_VEL
LIN {X 0,Y 413.786,Z 490.698,A -85,B 0,C 180,E1 -10671.465,E2 -10671.465} C_VEL
LIN {X 0,Y 412.99,Z 500.542,A -85,B 0,C 180,E1 -10672.498,E2 -10672.498} C_VEL
LIN {X 0,Y 412.446,Z 507.689,A -85,B 0,C 180,E1 -10673.388,E2 -10673.388} C_VEL
LIN {X 0,Y 411.82,Z 515.403,A -85,B 0,C 180,E1 -10674.533,E2 -10674.533} C_VEL
LIN {X 0,Y 411.172,Z 523.245,A -85,B 0,C 180,E1 -10675.959,E2 -10675.959} C_VEL
LIN {X 0,Y 410.878,Z 527.875,A -85,B 0,C 180,E1 -10676.944,E2 -10676.944} C_VEL
LIN {X 0,Y 410.444,Z 533.676,A -85,B 0,C 180,E1 -10678.469,E2 -10678.469} C_VEL
LIN {X 0,Y 410.251,Z 537.284,A -85,B 0,C 180,E1 -10679.645,E2 -10679.645} C_VEL
LIN {X 0,Y 409.999,Z 541.255,A -85,B 0,C 180,E1 -10681.317,E2 -10681.317} C_VEL
LIN {X 0,Y 409.78,Z 544.028,A -85,B 0,C 180,E1 -10683.105,E2 -10683.105} C_VEL
LIN {X 0,Y 409.666,Z 545.359,A -85,B 0,C 180,E1 -10684.603,E2 -10684.603} C_VEL
LIN {X 0,Y 409.676,Z 545.707,A -85,B 0,C 180,E1 -10685.687,E2 -10685.687} C_VEL
LIN {X 0,Y 409.716,Z 545.034,A -85,B 0,C 180,E1 -10687.829,E2 -10687.829} C_VEL
LIN {X 0,Y 409.777,Z 543.99,A -85,B 0,C 180,E1 -10688.89,E2 -10688.89} C_VEL
LIN {X 0,Y 409.981,Z 541.452,A -85,B 0,C 180,E1 -10690.531,E2 -10690.531} C_VEL
LIN {X 0,Y 410.174,Z 538.034,A -85,B 0,C 180,E1 -10692.036,E2 -10692.036} C_VEL
LIN {X 0,Y 410.503,Z 532.543,A -85,B 0,C 180,E1 -10693.814,E2 -10693.814} C_VEL
LIN {X 0,Y 410.905,Z 526.133,A -85,B 0,C 180,E1 -10695.388,E2 -10695.388} C_VEL
LIN {X 0,Y 411.338,Z 520.375,A -85,B 0,C 180,E1 -10696.556,E2 -10696.556} C_VEL
LIN {X 0,Y 411.947,Z 512.023,A -85,B 0,C 180,E1 -10697.937,E2 -10697.937} C_VEL
LIN {X 0,Y 412.587,Z 504.006,A -85,B 0,C 180,E1 -10699.033,E2 -10699.033} C_VEL
LIN {X 0,Y 413.118,Z 496.007,A -85,B 0,C 180,E1 -10699.958,E2 -10699.958} C_VEL
LIN {X 0,Y 413.749,Z 488.213,A -85,B 0,C 180,E1 -10700.718,E2 -10700.718} C_VEL
LIN {X 0,Y 413.561,Z 483.22,A -85,B 0,C 180,E1 -10701.153,E2 -10701.153} C_VEL
LIN {X 0,Y 411.924,Z 476.646,A -85,B 0,C 180,E1 -10701.727,E2 -10701.727} C_VEL
LIN {X 0,Y 409.09,Z 466.516,A -85,B 0,C 180,E1 -10702.498,E2 -10702.498} C_VEL
LIN {X 0,Y 408.441,Z 461.088,A -85,B 0,C 180,E1 -10702.807,E2 -10702.807} C_VEL
LIN {X 0,Y 408.919,Z 448.826,A -85,B 0,C 180,E1 -10703.307,E2 -10703.307} C_VEL
LIN {X 0,Y 409.256,Z 433.359,A -85,B 0,C 180,E1 -10703.684,E2 -10703.684} C_VEL
LIN {X 0,Y 410.159,Z 356.651,A -85,B 0,C 180,E1 -10705.051,E2 -10705.051} C_VEL
LIN {X 0,Y 406.13,Z 335.258,A -85,B 0,C 180,E1 -10705.658,E2 -10705.658} C_VEL
LIN {X 0,Y 406.083,Z 334.356,A -85,B 0,C 180,E1 -10705.782,E2 -10705.782} C_VEL
LIN {X 0,Y 406.674,Z 325.784,A -85,B 0,C 180,E1 -10707.772,E2 -10707.772} C_VEL
LIN {X 0,Y 404.97,Z 314.941,A -85,B 0,C 180,E1 -10710.497,E2 -10710.497} C_VEL
LIN {X 0,Y 404.429,Z 312.665,A -85,B 0,C 180,E1 -10711.151,E2 -10711.151} C_VEL
LIN {X 0,Y 404.423,Z 312.61,A -85,B 0,C 180,E1 -10712.988,E2 -10712.988} C_VEL
LIN {X 0,Y 404.415,Z 312.604,A -85,B 0,C 180,E1 -10715.985,E2 -10715.985} C_VEL
LIN {X 0,Y 404.268,Z 312.623,A -85,B 0,C 180,E1 -10719.002,E2 -10719.002} C_VEL
LIN {X 0,Y 404.258,Z 312.624,A -85,B 0,C 180,E1 -10722.042,E2 -10722.042} C_VEL
LIN {X 0,Y 404.208,Z 312.63,A -85,B 0,C 180,E1 -10725.118,E2 -10725.118} C_VEL
LIN {X 0,Y 404.212,Z 312.632,A -85,B 0,C 180,E1 -10728.238,E2 -10728.238} C_VEL
LIN {X 0,Y 404.14,Z 312.64,A -85,B 0,C 180,E1 -10731.419,E2 -10731.419} C_VEL
LIN {X 0,Y 404.176,Z 312.638,A -85,B 0,C 180,E1 -10734.666,E2 -10734.666} C_VEL
LIN {X 0,Y 404.197,Z 312.625,A -85,B 0,C 180,E1 -10738,E2 -10738} C_VEL
LIN {X 0,Y 404.141,Z 312.642,A -85,B 0,C 180,E1 -10741.558,E2 -10741.558} C_VEL
LIN {X 0,Y 404.186,Z 312.624,A -85,B 0,C 180,E1 -10745.016,E2 -10745.016} C_VEL
LIN {X 0,Y 404.159,Z 312.636,A -85,B 0,C 180,E1 -10748.757,E2 -10748.757} C_VEL
LIN {X 0,Y 404.125,Z 312.632,A -85,B 0,C 180,E1 -10751.6,E2 -10751.6} C_VEL
LIN {X 0,Y 404.147,Z 312.643,A -85,B 0,C 180,E1 -10754.522,E2 -10754.522} C_VEL
LIN {X 0,Y 404.134,Z 312.638,A -85,B 0,C 180,E1 -10757.295,E2 -10757.295} C_VEL
LIN {X 0,Y 404.136,Z 312.624,A -85,B 0,C 180,E1 -10759.951,E2 -10759.951} C_VEL
LIN {X 0,Y 404.137,Z 312.638,A -85,B 0,C 180,E1 -10763.125,E2 -10763.125} C_VEL
LIN {X 0,Y 404.146,Z 312.637,A -85,B 0,C 180,E1 -10766.188,E2 -10766.188} C_VEL
LIN {X 0,Y 404.146,Z 312.623,A -85,B 0,C 180,E1 -10769.715,E2 -10769.715} C_VEL
LIN {X 0,Y 404.137,Z 312.631,A -85,B 0,C 180,E1 -10773.118,E2 -10773.118} C_VEL
LIN {X 0,Y 404.168,Z 312.641,A -85,B 0,C 180,E1 -10776.425,E2 -10776.425} C_VEL
LIN {X 0,Y 404.194,Z 312.623,A -85,B 0,C 180,E1 -10779.874,E2 -10779.874} C_VEL
LIN {X 0,Y 404.218,Z 312.613,A -85,B 0,C 180,E1 -10782.993,E2 -10782.993} C_VEL
LIN {X 0,Y 404.285,Z 312.622,A -85,B 0,C 180,E1 -10786.939,E2 -10786.939} C_VEL
LIN {X 0,Y 404.256,Z 312.62,A -85,B 0,C 180,E1 -10789.988,E2 -10789.988} C_VEL
LIN {X 0,Y 404.343,Z 312.594,A -85,B 0,C 180,E1 -10793.011,E2 -10793.011} C_VEL
LIN {X 0,Y 404.265,Z 312.607,A -85,B 0,C 180,E1 -10795.013,E2 -10795.013} C_VEL
LIN {X 0,Y 404.474,Z 312.598,A -85,B 0,C 180,E1 -10798.008,E2 -10798.008} C_VEL
LIN {X 0,Y 404.403,Z 312.603,A -85,B 0,C 180,E1 -10800.996,E2 -10800.996} C_VEL
LIN {X 0,Y 404.389,Z 312.596,A -85,B 0,C 180,E1 -10802.988,E2 -10802.988} C_VEL
LIN {X 0,Y 404.384,Z 312.602,A -85,B 0,C 180,E1 -10806.987,E2 -10806.987} C_VEL
LIN {X 0,Y 404.251,Z 312.629,A -85,B 0,C 180,E1 -10811.025,E2 -10811.025} C_VEL
LIN {X 0,Y 404.268,Z 312.622,A -85,B 0,C 180,E1 -10813.211,E2 -10813.211} C_VEL
LIN {X 0,Y 404.177,Z 312.628,A -85,B 0,C 180,E1 -10817.193,E2 -10817.193} C_VEL
LIN {X 0,Y 404.165,Z 312.64,A -85,B 0,C 180,E1 -10820.351,E2 -10820.351} C_VEL
LIN {X 0,Y 404.149,Z 312.625,A -85,B 0,C 180,E1 -10823.575,E2 -10823.575} C_VEL
LIN {X 0,Y 404.106,Z 312.65,A -85,B 0,C 180,E1 -10826.883,E2 -10826.883} C_VEL
LIN {X 0,Y 404.143,Z 312.634,A -85,B 0,C 180,E1 -10830.285,E2 -10830.285} C_VEL
LIN {X 0,Y 404.137,Z 312.643,A -85,B 0,C 180,E1 -10833.813,E2 -10833.813} C_VEL
LIN {X 0,Y 404.132,Z 312.636,A -85,B 0,C 180,E1 -10836.874,E2 -10836.874} C_VEL
LIN {X 0,Y 404.116,Z 312.648,A -85,B 0,C 180,E1 -10840.074,E2 -10840.074} C_VEL
LIN {X 0,Y 404.139,Z 312.636,A -85,B 0,C 180,E1 -10843.081,E2 -10843.081} C_VEL
LIN {X 0,Y 404.118,Z 312.644,A -85,B 0,C 180,E1 -10845.922,E2 -10845.922} C_VEL
LIN {X 0,Y 404.1,Z 312.65,A -85,B 0,C 180,E1 -10848.632,E2 -10848.632} C_VEL
LIN {X 0,Y 404.138,Z 312.641,A -85,B 0,C 180,E1 -10851.495,E2 -10851.495} C_VEL
LIN {X 0,Y 404.172,Z 312.641,A -85,B 0,C 180,E1 -10854.982,E2 -10854.982} C_VEL
LIN {X 0,Y 404.136,Z 312.642,A -85,B 0,C 180,E1 -10858.442,E2 -10858.442} C_VEL
LIN {X 0,Y 404.155,Z 312.642,A -85,B 0,C 180,E1 -10860.863,E2 -10860.863} C_VEL
LIN {X 0,Y 404.169,Z 312.742,A -85,B 0,C 180,E1 -10862.918,E2 -10862.918} C_VEL
LIN {X 0,Y 405.781,Z 320.672,A -85,B 0,C 180,E1 -10864.891,E2 -10864.891} C_VEL
LIN {X 0,Y 407.067,Z 327.935,A -85,B 0,C 180,E1 -10866.603,E2 -10866.603} C_VEL
LIN {X 0,Y 406.074,Z 342.38,A -85,B 0,C 180,E1 -10869.748,E2 -10869.748} C_VEL
LIN {X 0,Y 405.904,Z 345.436,A -85,B 0,C 180,E1 -10870.35,E2 -10870.35} C_VEL
LIN {X 0,Y 410.106,Z 370.468,A -85,B 0,C 180,E1 -10871.039,E2 -10871.039} C_VEL
LIN {X 0,Y 409.162,Z 451.293,A -85,B 0,C 180,E1 -10872.507,E2 -10872.507} C_VEL
LIN {X 0,Y 408.846,Z 461.176,A -85,B 0,C 180,E1 -10872.783,E2 -10872.783} C_VEL
LIN {X 0,Y 408.292,Z 471.169,A -85,B 0,C 180,E1 -10873.178,E2 -10873.178} C_VEL
LIN {X 0,Y 407.825,Z 481.535,A -85,B 0,C 180,E1 -10873.738,E2 -10873.738} C_VEL
LIN {X 0,Y 407.098,Z 492.23,A -85,B 0,C 180,E1 -10874.479,E2 -10874.479} C_VEL
LIN {X 0,Y 406.389,Z 502.434,A -85,B 0,C 180,E1 -10875.37,E2 -10875.37} C_VEL
LIN {X 0,Y 405.698,Z 511.6,A -85,B 0,C 180,E1 -10876.348,E2 -10876.348} C_VEL
LIN {X 0,Y 405.04,Z 520.308,A -85,B 0,C 180,E1 -10877.473,E2 -10877.473} C_VEL
LIN {X 0,Y 404.496,Z 526.892,A -85,B 0,C 180,E1 -10878.474,E2 -10878.474} C_VEL
LIN {X 0,Y 403.973,Z 533.801,A -85,B 0,C 180,E1 -10879.728,E2 -10879.728} C_VEL
LIN {X 0,Y 403.565,Z 539.579,A -85,B 0,C 180,E1 -10880.983,E2 -10880.983} C_VEL
LIN {X 0,Y 403.206,Z 545.172,A -85,B 0,C 180,E1 -10882.488,E2 -10882.488} C_VEL
LIN {X 0,Y 402.983,Z 549.574,A -85,B 0,C 180,E1 -10883.993,E2 -10883.993} C_VEL
LIN {X 0,Y 402.944,Z 551.892,A -85,B 0,C 180,E1 -10884.997,E2 -10884.997} C_VEL
LIN {X 0,Y 402.78,Z 555.25,A -85,B 0,C 180,E1 -10886.999,E2 -10886.999} C_VEL
LIN {X 0,Y 402.84,Z 556.832,A -85,B 0,C 180,E1 -10889,E2 -10889} C_VEL
LIN {X 0,Y 402.826,Z 557.141,A -85,B 0,C 180,E1 -10890,E2 -10890} C_VEL
LIN {X 0,Y 402.817,Z 556.332,A -85,B 0,C 180,E1 -10892,E2 -10892} C_VEL
LIN {X 0,Y 402.78,Z 555.359,A -85,B 0,C 180,E1 -10893,E2 -10893} C_VEL
LIN {X 0,Y 402.966,Z 552.171,A -85,B 0,C 180,E1 -10895.003,E2 -10895.003} C_VEL
LIN {X 0,Y 403.047,Z 548.598,A -85,B 0,C 180,E1 -10896.507,E2 -10896.507} C_VEL
LIN {X 0,Y 403.314,Z 543.908,A -85,B 0,C 180,E1 -10898.013,E2 -10898.013} C_VEL
LIN {X 0,Y 403.709,Z 537.955,A -85,B 0,C 180,E1 -10899.519,E2 -10899.519} C_VEL
LIN {X 0,Y 404.217,Z 531.941,A -85,B 0,C 180,E1 -10900.772,E2 -10900.772} C_VEL
LIN {X 0,Y 404.826,Z 524.687,A -85,B 0,C 180,E1 -10902.024,E2 -10902.024} C_VEL
LIN {X 0,Y 405.611,Z 515.865,A -85,B 0,C 180,E1 -10903.272,E2 -10903.272} C_VEL
LIN {X 0,Y 406.253,Z 506.595,A -85,B 0,C 180,E1 -10904.357,E2 -10904.357} C_VEL
LIN {X 0,Y 406.97,Z 497.098,A -85,B 0,C 180,E1 -10905.269,E2 -10905.269} C_VEL
LIN {X 0,Y 407.661,Z 487.652,A -85,B 0,C 180,E1 -10906.012,E2 -10906.012} C_VEL
LIN {X 0,Y 408.407,Z 476.727,A -85,B 0,C 180,E1 -10906.688,E2 -10906.688} C_VEL
LIN {X 0,Y 408.952,Z 465.581,A -85,B 0,C 180,E1 -10907.212,E2 -10907.212} C_VEL
LIN {X 0,Y 409.388,Z 455.696,A -85,B 0,C 180,E1 -10907.547,E2 -10907.547} C_VEL
LIN {X 0,Y 409.681,Z 441.278,A -85,B 0,C 180,E1 -10907.857,E2 -10907.857} C_VEL
LIN {X 0,Y 410.512,Z 370.745,A -85,B 0,C 180,E1 -10909.125,E2 -10909.125} C_VEL
LIN {X 0,Y 406.207,Z 345.889,A -85,B 0,C 180,E1 -10909.828,E2 -10909.828} C_VEL
LIN {X 0,Y 406.08,Z 344.829,A -85,B 0,C 180,E1 -10909.897,E2 -10909.897} C_VEL
LIN {X 0,Y 407.133,Z 329.471,A -85,B 0,C 180,E1 -10913.123,E2 -10913.123} C_VEL
LIN {X 0,Y 406.563,Z 324.325,A -85,B 0,C 180,E1 -10914.289,E2 -10914.289} C_VEL
LIN {X 0,Y 404.178,Z 312.774,A -85,B 0,C 180,E1 -10917.081,E2 -10917.081} C_VEL
LIN {X 0,Y 404.142,Z 312.644,A -85,B 0,C 180,E1 -10920.285,E2 -10920.285} C_VEL
LIN {X 0,Y 404.142,Z 312.64,A -85,B 0,C 180,E1 -10923.812,E2 -10923.812} C_VEL
LIN {X 0,Y 404.134,Z 312.64,A -85,B 0,C 180,E1 -10926.875,E2 -10926.875} C_VEL
LIN {X 0,Y 404.146,Z 312.634,A -85,B 0,C 180,E1 -10930.08,E2 -10930.08} C_VEL
LIN {X 0,Y 404.148,Z 312.643,A -85,B 0,C 180,E1 -10933.084,E2 -10933.084} C_VEL
LIN {X 0,Y 404.146,Z 312.64,A -85,B 0,C 180,E1 -10935.926,E2 -10935.926} C_VEL
LIN {X 0,Y 404.117,Z 312.639,A -85,B 0,C 180,E1 -10938.635,E2 -10938.635} C_VEL
LIN {X 0,Y 404.149,Z 312.641,A -85,B 0,C 180,E1 -10941.493,E2 -10941.493} C_VEL
LIN {X 0,Y 404.184,Z 312.63,A -85,B 0,C 180,E1 -10944.984,E2 -10944.984} C_VEL
LIN {X 0,Y 404.141,Z 312.639,A -85,B 0,C 180,E1 -10948.554,E2 -10948.554} C_VEL
LIN {X 0,Y 404.195,Z 312.634,A -85,B 0,C 180,E1 -10952.001,E2 -10952.001} C_VEL
LIN {X 0,Y 404.177,Z 312.635,A -85,B 0,C 180,E1 -10955.335,E2 -10955.335} C_VEL
LIN {X 0,Y 404.139,Z 312.64,A -85,B 0,C 180,E1 -10958.581,E2 -10958.581} C_VEL
LIN {X 0,Y 404.211,Z 312.629,A -85,B 0,C 180,E1 -10961.762,E2 -10961.762} C_VEL
LIN {X 0,Y 404.208,Z 312.632,A -85,B 0,C 180,E1 -10964.882,E2 -10964.882} C_VEL
LIN {X 0,Y 404.258,Z 312.63,A -85,B 0,C 180,E1 -10967.959,E2 -10967.959} C_VEL
LIN {X 0,Y 404.434,Z 312.604,A -85,B 0,C 180,E1 -10972.1,E2 -10972.1} C_VEL
LIN {X 0,Y 404.426,Z 312.611,A -85,B 0,C 180,E1 -10974.015,E2 -10974.015} C_VEL
LIN {X 0,Y 404.484,Z 312.599,A -85,B 0,C 180,E1 -10978.009,E2 -10978.009} C_VEL
LIN {X 0,Y 404.613,Z 312.579,A -85,B 0,C 180,E1 -10980,E2 -10980} C_VEL
LIN {X 0,Y 404.424,Z 312.608,A -85,B 0,C 180,E1 -10982.989,E2 -10982.989} C_VEL
LIN {X 0,Y 404.414,Z 312.612,A -85,B 0,C 180,E1 -10986.987,E2 -10986.987} C_VEL
LIN {X 0,Y 404.26,Z 312.625,A -85,B 0,C 180,E1 -10990.012,E2 -10990.012} C_VEL
LIN {X 0,Y 404.268,Z 312.623,A -85,B 0,C 180,E1 -10993.212,E2 -10993.212} C_VEL
LIN {X 0,Y 404.217,Z 312.63,A -85,B 0,C 180,E1 -10997.007,E2 -10997.007} C_VEL
LIN {X 0,Y 404.165,Z 312.641,A -85,B 0,C 180,E1 -11000.352,E2 -11000.352} C_VEL
LIN {X 0,Y 404.161,Z 312.639,A -85,B 0,C 180,E1 -11003.575,E2 -11003.575} C_VEL
LIN {X 0,Y 404.167,Z 312.632,A -85,B 0,C 180,E1 -11006.879,E2 -11006.879} C_VEL
LIN {X 0,Y 404.146,Z 312.643,A -85,B 0,C 180,E1 -11010.285,E2 -11010.285} C_VEL
LIN {X 0,Y 404.145,Z 312.637,A -85,B 0,C 180,E1 -11013.812,E2 -11013.812} C_VEL
LIN {X 0,Y 404.137,Z 312.642,A -85,B 0,C 180,E1 -11016.875,E2 -11016.875} C_VEL
LIN {X 0,Y 404.148,Z 312.643,A -85,B 0,C 180,E1 -11020.08,E2 -11020.08} C_VEL
LIN {X 0,Y 404.184,Z 312.851,A -85,B 0,C 180,E1 -11021.357,E2 -11021.357} C_VEL
LIN {X 0,Y 406.513,Z 324.17,A -85,B 0,C 180,E1 -11024.031,E2 -11024.031} C_VEL
LIN {X 0,Y 406.352,Z 332.173,A -85,B 0,C 180,E1 -11025.747,E2 -11025.747} C_VEL
LIN {X 0,Y 406.306,Z 334.619,A -85,B 0,C 180,E1 -11026.188,E2 -11026.188} C_VEL
LIN {X 0,Y 410.416,Z 355.857,A -85,B 0,C 180,E1 -11026.835,E2 -11026.835} C_VEL
LIN {X 0,Y 410.707,Z 359.931,A -85,B 0,C 180,E1 -11026.926,E2 -11026.926} C_VEL
LIN {X 0,Y 409.457,Z 440.648,A -85,B 0,C 180,E1 -11028.392,E2 -11028.392} C_VEL
LIN {X 0,Y 409.183,Z 450.807,A -85,B 0,C 180,E1 -11028.686,E2 -11028.686} C_VEL
LIN {X 0,Y 408.844,Z 460.209,A -85,B 0,C 180,E1 -11029.069,E2 -11029.069} C_VEL
LIN {X 0,Y 408.272,Z 470.659,A -85,B 0,C 180,E1 -11029.633,E2 -11029.633} C_VEL
LIN {X 0,Y 407.613,Z 481.1,A -85,B 0,C 180,E1 -11030.361,E2 -11030.361} C_VEL
LIN {X 0,Y 406.989,Z 490.097,A -85,B 0,C 180,E1 -11031.132,E2 -11031.132} C_VEL
LIN {X 0,Y 406.09,Z 500.618,A -85,B 0,C 180,E1 -11032.25,E2 -11032.25} C_VEL
LIN {X 0,Y 405.437,Z 508.564,A -85,B 0,C 180,E1 -11033.271,E2 -11033.271} C_VEL
LIN {X 0,Y 404.872,Z 515.558,A -85,B 0,C 180,E1 -11034.332,E2 -11034.332} C_VEL
LIN {X 0,Y 404.259,Z 522.528,A -85,B 0,C 180,E1 -11035.597,E2 -11035.597} C_VEL
LIN {X 0,Y 403.782,Z 528.807,A -85,B 0,C 180,E1 -11036.986,E2 -11036.986} C_VEL
LIN {X 0,Y 403.336,Z 534.693,A -85,B 0,C 180,E1 -11038.629,E2 -11038.629} C_VEL
LIN {X 0,Y 403.174,Z 537.709,A -85,B 0,C 180,E1 -11039.634,E2 -11039.634} C_VEL
LIN {X 0,Y 402.918,Z 541.557,A -85,B 0,C 180,E1 -11041.336,E2 -11041.336} C_VEL
LIN {X 0,Y 402.71,Z 544.103,A -85,B 0,C 180,E1 -11043.016,E2 -11043.016} C_VEL
LIN {X 0,Y 402.604,Z 545.164,A -85,B 0,C 180,E1 -11044.125,E2 -11044.125} C_VEL
LIN {X 0,Y 402.583,Z 545.668,A -85,B 0,C 180,E1 -11045.23,E2 -11045.23} C_VEL
LIN {X 0,Y 402.56,Z 545.792,A -85,B 0,C 180,E1 -11046.326,E2 -11046.326} C_VEL
LIN {X 0,Y 402.605,Z 545.276,A -85,B 0,C 180,E1 -11047.696,E2 -11047.696} C_VEL
LIN {X 0,Y 402.752,Z 543.211,A -85,B 0,C 180,E1 -11049.574,E2 -11049.574} C_VEL
LIN {X 0,Y 402.965,Z 540.325,A -85,B 0,C 180,E1 -11051.177,E2 -11051.177} C_VEL
LIN {X 0,Y 403.124,Z 537.872,A -85,B 0,C 180,E1 -11052.236,E2 -11052.236} C_VEL
LIN {X 0,Y 403.42,Z 533.088,A -85,B 0,C 180,E1 -11053.815,E2 -11053.815} C_VEL
LIN {X 0,Y 403.834,Z 526.949,A -85,B 0,C 180,E1 -11055.384,E2 -11055.384} C_VEL
LIN {X 0,Y 404.332,Z 520.335,A -85,B 0,C 180,E1 -11056.75,E2 -11056.75} C_VEL
LIN {X 0,Y 404.883,Z 513.161,A -85,B 0,C 180,E1 -11057.978,E2 -11057.978} C_VEL
LIN {X 0,Y 405.655,Z 503.926,A -85,B 0,C 180,E1 -11059.266,E2 -11059.266} C_VEL
LIN {X 0,Y 406.227,Z 496.016,A -85,B 0,C 180,E1 -11060.193,E2 -11060.193} C_VEL
LIN {X 0,Y 406.948,Z 487.139,A -85,B 0,C 180,E1 -11061.058,E2 -11061.058} C_VEL
LIN {X 0,Y 407.542,Z 477.691,A -85,B 0,C 180,E1 -11061.821,E2 -11061.821} C_VEL
LIN {X 0,Y 408.15,Z 466.752,A -85,B 0,C 180,E1 -11062.518,E2 -11062.518} C_VEL
LIN {X 0,Y 408.441,Z 461.088,A -85,B 0,C 180,E1 -11062.807,E2 -11062.807} C_VEL
LIN {X 0,Y 408.014,Z 455.546,A -85,B 0,C 180,E1 -11063.094,E2 -11063.094} C_VEL
LIN {X 0,Y 405.546,Z 446.441,A -85,B 0,C 180,E1 -11063.534,E2 -11063.534} C_VEL
LIN {X 0,Y 403.036,Z 437.167,A -85,B 0,C 180,E1 -11063.878,E2 -11063.878} C_VEL
LIN {X 0,Y 402.523,Z 431.365,A -85,B 0,C 180,E1 -11064.013,E2 -11064.013} C_VEL
LIN {X 0,Y 403.423,Z 357.721,A -85,B 0,C 180,E1 -11065.348,E2 -11065.348} C_VEL
LIN {X 0,Y 399.204,Z 335.335,A -85,B 0,C 180,E1 -11065.994,E2 -11065.994} C_VEL
LIN {X 0,Y 399.253,Z 333.974,A -85,B 0,C 180,E1 -11066.215,E2 -11066.215} C_VEL
LIN {X 0,Y 399.674,Z 326.575,A -85,B 0,C 180,E1 -11067.985,E2 -11067.985} C_VEL
LIN {X 0,Y 398.11,Z 316.725,A -85,B 0,C 180,E1 -11070.506,E2 -11070.506} C_VEL
LIN {X 0,Y 397.418,Z 313.513,A -85,B 0,C 180,E1 -11071.425,E2 -11071.425} C_VEL
LIN {X 0,Y 397.382,Z 313.487,A -85,B 0,C 180,E1 -11073.041,E2 -11073.041} C_VEL
LIN {X 0,Y 397.366,Z 313.482,A -85,B 0,C 180,E1 -11076.092,E2 -11076.092} C_VEL
LIN {X 0,Y 397.238,Z 313.5,A -85,B 0,C 180,E1 -11079.162,E2 -11079.162} C_VEL
LIN {X 0,Y 397.221,Z 313.5,A -85,B 0,C 180,E1 -11082.258,E2 -11082.258} C_VEL
LIN {X 0,Y 397.181,Z 313.507,A -85,B 0,C 180,E1 -11085.392,E2 -11085.392} C_VEL
LIN {X 0,Y 397.164,Z 313.506,A -85,B 0,C 180,E1 -11088.573,E2 -11088.573} C_VEL
LIN {X 0,Y 397.098,Z 313.518,A -85,B 0,C 180,E1 -11091.819,E2 -11091.819} C_VEL
LIN {X 0,Y 397.154,Z 313.511,A -85,B 0,C 180,E1 -11095.512,E2 -11095.512} C_VEL
LIN {X 0,Y 397.124,Z 313.508,A -85,B 0,C 180,E1 -11098.544,E2 -11098.544} C_VEL
LIN {X 0,Y 397.08,Z 313.518,A -85,B 0,C 180,E1 -11102.072,E2 -11102.072} C_VEL
LIN {X 0,Y 397.12,Z 313.509,A -85,B 0,C 180,E1 -11105.503,E2 -11105.503} C_VEL
LIN {X 0,Y 397.134,Z 313.511,A -85,B 0,C 180,E1 -11108.862,E2 -11108.862} C_VEL
LIN {X 0,Y 397.07,Z 313.512,A -85,B 0,C 180,E1 -11112.267,E2 -11112.267} C_VEL
LIN {X 0,Y 397.088,Z 313.519,A -85,B 0,C 180,E1 -11115.069,E2 -11115.069} C_VEL
LIN {X 0,Y 397.063,Z 313.518,A -85,B 0,C 180,E1 -11118.022,E2 -11118.022} C_VEL
LIN {X 0,Y 397.105,Z 313.504,A -85,B 0,C 180,E1 -11121.143,E2 -11121.143} C_VEL
LIN {X 0,Y 397.121,Z 313.512,A -85,B 0,C 180,E1 -11124.497,E2 -11124.497} C_VEL
LIN {X 0,Y 397.08,Z 313.512,A -85,B 0,C 180,E1 -11127.928,E2 -11127.928} C_VEL
LIN {X 0,Y 397.12,Z 313.492,A -85,B 0,C 180,E1 -11130.295,E2 -11130.295} C_VEL
LIN {X 0,Y 397.097,Z 313.512,A -85,B 0,C 180,E1 -11133.739,E2 -11133.739} C_VEL
LIN {X 0,Y 397.11,Z 313.514,A -85,B 0,C 180,E1 -11137.086,E2 -11137.086} C_VEL
LIN {X 0,Y 397.148,Z 313.499,A -85,B 0,C 180,E1 -11140.353,E2 -11140.353} C_VEL
LIN {X 0,Y 397.168,Z 313.497,A -85,B 0,C 180,E1 -11143.553,E2 -11143.553} C_VEL
LIN {X 0,Y 397.231,Z 313.499,A -85,B 0,C 180,E1 -11146.703,E2 -11146.703} C_VEL
LIN {X 0,Y 397.216,Z 313.499,A -85,B 0,C 180,E1 -11149.809,E2 -11149.809} C_VEL
LIN {X 0,Y 397.295,Z 313.471,A -85,B 0,C 180,E1 -11152.887,E2 -11152.887} C_VEL
LIN {X 0,Y 397.236,Z 313.482,A -85,B 0,C 180,E1 -11154.925,E2 -11154.925} C_VEL
LIN {X 0,Y 397.443,Z 313.473,A -85,B 0,C 180,E1 -11157.973,E2 -11157.973} C_VEL
LIN {X 0,Y 397.369,Z 313.479,A -85,B 0,C 180,E1 -11161.013,E2 -11161.013} C_VEL
LIN {X 0,Y 397.324,Z 313.475,A -85,B 0,C 180,E1 -11163.042,E2 -11163.042} C_VEL
LIN {X 0,Y 397.35,Z 313.469,A -85,B 0,C 180,E1 -11166.092,E2 -11166.092} C_VEL
LIN {X 0,Y 397.236,Z 313.503,A -85,B 0,C 180,E1 -11169.162,E2 -11169.162} C_VEL
LIN {X 0,Y 397.22,Z 313.497,A -85,B 0,C 180,E1 -11172.258,E2 -11172.258} C_VEL
LIN {X 0,Y 397.123,Z 313.498,A -85,B 0,C 180,E1 -11175.394,E2 -11175.394} C_VEL
LIN {X 0,Y 397.112,Z 313.516,A -85,B 0,C 180,E1 -11178.576,E2 -11178.576} C_VEL
LIN {X 0,Y 397.096,Z 313.517,A -85,B 0,C 180,E1 -11181.818,E2 -11181.818} C_VEL
LIN {X 0,Y 397.097,Z 313.514,A -85,B 0,C 180,E1 -11185.135,E2 -11185.135} C_VEL
LIN {X 0,Y 397.065,Z 313.524,A -85,B 0,C 180,E1 -11188.548,E2 -11188.548} C_VEL
LIN {X 0,Y 397.08,Z 313.514,A -85,B 0,C 180,E1 -11191.836,E2 -11191.836} C_VEL
LIN {X 0,Y 397.119,Z 313.514,A -85,B 0,C 180,E1 -11194.494,E2 -11194.494} C_VEL
LIN {X 0,Y 397.09,Z 313.518,A -85,B 0,C 180,E1 -11198.276,E2 -11198.276} C_VEL
LIN {X 0,Y 397.049,Z 313.523,A -85,B 0,C 180,E1 -11201.976,E2 -11201.976} C_VEL
LIN {X 0,Y 397.082,Z 313.519,A -85,B 0,C 180,E1 -11205.069,E2 -11205.069} C_VEL
LIN {X 0,Y 397.049,Z 313.525,A -85,B 0,C 180,E1 -11208.023,E2 -11208.023} C_VEL
LIN {X 0,Y 397.09,Z 313.518,A -85,B 0,C 180,E1 -11211.723,E2 -11211.723} C_VEL
LIN {X 0,Y 397.115,Z 313.514,A -85,B 0,C 180,E1 -11215.506,E2 -11215.506} C_VEL
LIN {X 0,Y 397.075,Z 313.521,A -85,B 0,C 180,E1 -11219.117,E2 -11219.117} C_VEL
LIN {X 0,Y 397.129,Z 313.661,A -85,B 0,C 180,E1 -11222.676,E2 -11222.676} C_VEL
LIN {X 0,Y 399.228,Z 324.128,A -85,B 0,C 180,E1 -11225.286,E2 -11225.286} C_VEL
LIN {X 0,Y 400.115,Z 330.167,A -85,B 0,C 180,E1 -11226.721,E2 -11226.721} C_VEL
LIN {X 0,Y 398.996,Z 345.036,A -85,B 0,C 180,E1 -11229.978,E2 -11229.978} C_VEL
LIN {X 0,Y 399.386,Z 347.716,A -85,B 0,C 180,E1 -11230.111,E2 -11230.111} C_VEL
LIN {X 0,Y 403.38,Z 371.971,A -85,B 0,C 180,E1 -11230.758,E2 -11230.758} C_VEL
LIN {X 0,Y 402.346,Z 450.581,A -85,B 0,C 180,E1 -11232.201,E2 -11232.201} C_VEL
LIN {X 0,Y 402.031,Z 461.515,A -85,B 0,C 180,E1 -11232.515,E2 -11232.515} C_VEL
LIN {X 0,Y 401.424,Z 471.993,A -85,B 0,C 180,E1 -11232.947,E2 -11232.947} C_VEL
LIN {X 0,Y 400.996,Z 481.214,A -85,B 0,C 180,E1 -11233.453,E2 -11233.453} C_VEL
LIN {X 0,Y 400.249,Z 491.953,A -85,B 0,C 180,E1 -11234.207,E2 -11234.207} C_VEL
LIN {X 0,Y 399.483,Z 502.361,A -85,B 0,C 180,E1 -11235.129,E2 -11235.129} C_VEL
LIN {X 0,Y 398.786,Z 511.38,A -85,B 0,C 180,E1 -11236.106,E2 -11236.106} C_VEL
LIN {X 0,Y 398.095,Z 520.109,A -85,B 0,C 180,E1 -11237.251,E2 -11237.251} C_VEL
LIN {X 0,Y 397.512,Z 526.71,A -85,B 0,C 180,E1 -11238.269,E2 -11238.269} C_VEL
LIN {X 0,Y 396.973,Z 533.634,A -85,B 0,C 180,E1 -11239.545,E2 -11239.545} C_VEL
LIN {X 0,Y 396.525,Z 539.425,A -85,B 0,C 180,E1 -11240.821,E2 -11240.821} C_VEL
LIN {X 0,Y 396.155,Z 545.03,A -85,B 0,C 180,E1 -11242.354,E2 -11242.354} C_VEL
LIN {X 0,Y 395.906,Z 549.443,A -85,B 0,C 180,E1 -11243.886,E2 -11243.886} C_VEL
LIN {X 0,Y 395.859,Z 551.761,A -85,B 0,C 180,E1 -11244.907,E2 -11244.907} C_VEL
LIN {X 0,Y 395.686,Z 555.138,A -85,B 0,C 180,E1 -11246.945,E2 -11246.945} C_VEL
LIN {X 0,Y 395.751,Z 556.729,A -85,B 0,C 180,E1 -11248.982,E2 -11248.982} C_VEL
LIN {X 0,Y 395.755,Z 557.04,A -85,B 0,C 180,E1 -11250,E2 -11250} C_VEL
LIN {X 0,Y 395.714,Z 556.244,A -85,B 0,C 180,E1 -11252.036,E2 -11252.036} C_VEL
LIN {X 0,Y 395.687,Z 555.27,A -85,B 0,C 180,E1 -11253.054,E2 -11253.054} C_VEL
LIN {X 0,Y 395.882,Z 552.097,A -85,B 0,C 180,E1 -11255.092,E2 -11255.092} C_VEL
LIN {X 0,Y 395.97,Z 548.531,A -85,B 0,C 180,E1 -11256.624,E2 -11256.624} C_VEL
LIN {X 0,Y 396.256,Z 543.849,A -85,B 0,C 180,E1 -11258.157,E2 -11258.157} C_VEL
LIN {X 0,Y 396.69,Z 537.905,A -85,B 0,C 180,E1 -11259.689,E2 -11259.689} C_VEL
LIN {X 0,Y 397.273,Z 530.476,A -85,B 0,C 180,E1 -11261.221,E2 -11261.221} C_VEL
LIN {X 0,Y 398.028,Z 522.956,A -85,B 0,C 180,E1 -11262.492,E2 -11262.492} C_VEL
LIN {X 0,Y 398.749,Z 514.84,A -85,B 0,C 180,E1 -11263.635,E2 -11263.635} C_VEL
LIN {X 0,Y 399.297,Z 507.465,A -85,B 0,C 180,E1 -11264.523,E2 -11264.523} C_VEL
LIN {X 0,Y 400.111,Z 497.162,A -85,B 0,C 180,E1 -11265.537,E2 -11265.537} C_VEL
LIN {X 0,Y 400.863,Z 487.767,A -85,B 0,C 180,E1 -11266.291,E2 -11266.291} C_VEL
LIN {X 0,Y 401.622,Z 476.909,A -85,B 0,C 180,E1 -11266.979,E2 -11266.979} C_VEL
LIN {X 0,Y 402.187,Z 465.871,A -85,B 0,C 180,E1 -11267.511,E2 -11267.511} C_VEL
LIN {X 0,Y 402.706,Z 454.922,A -85,B 0,C 180,E1 -11267.881,E2 -11267.881} C_VEL
LIN {X 0,Y 403.006,Z 438.521,A -85,B 0,C 180,E1 -11268.229,E2 -11268.229} C_VEL
LIN {X 0,Y 403.729,Z 370.775,A -85,B 0,C 180,E1 -11269.475,E2 -11269.475} C_VEL
LIN {X 0,Y 399.238,Z 345.141,A -85,B 0,C 180,E1 -11270.227,E2 -11270.227} C_VEL
LIN {X 0,Y 399.29,Z 343.004,A -85,B 0,C 180,E1 -11270.611,E2 -11270.611} C_VEL
LIN {X 0,Y 400.223,Z 329.456,A -85,B 0,C 180,E1 -11273.547,E2 -11273.547} C_VEL
LIN {X 0,Y 398.161,Z 318.378,A -85,B 0,C 180,E1 -11276.185,E2 -11276.185} C_VEL
LIN {X 0,Y 397.103,Z 313.591,A -85,B 0,C 180,E1 -11277.429,E2 -11277.429} C_VEL
LIN {X 0,Y 397.075,Z 313.524,A -85,B 0,C 180,E1 -11280.883,E2 -11280.883} C_VEL
LIN {X 0,Y 397.123,Z 313.516,A -85,B 0,C 180,E1 -11284.494,E2 -11284.494} C_VEL
LIN {X 0,Y 397.098,Z 313.519,A -85,B 0,C 180,E1 -11288.275,E2 -11288.275} C_VEL
LIN {X 0,Y 397.061,Z 313.519,A -85,B 0,C 180,E1 -11290.912,E2 -11290.912} C_VEL
LIN {X 0,Y 397.098,Z 313.521,A -85,B 0,C 180,E1 -11293.649,E2 -11293.649} C_VEL
LIN {X 0,Y 397.1,Z 313.517,A -85,B 0,C 180,E1 -11296.521,E2 -11296.521} C_VEL
LIN {X 0,Y 397.111,Z 313.516,A -85,B 0,C 180,E1 -11300.423,E2 -11300.423} C_VEL
LIN {X 0,Y 397.107,Z 313.515,A -85,B 0,C 180,E1 -11304.266,E2 -11304.266} C_VEL
LIN {X 0,Y 397.114,Z 313.517,A -85,B 0,C 180,E1 -11306.727,E2 -11306.727} C_VEL
LIN {X 0,Y 397.124,Z 313.518,A -85,B 0,C 180,E1 -11310.296,E2 -11310.296} C_VEL
LIN {X 0,Y 397.194,Z 313.504,A -85,B 0,C 180,E1 -11312.61,E2 -11312.61} C_VEL
LIN {X 0,Y 397.133,Z 313.511,A -85,B 0,C 180,E1 -11315.982,E2 -11315.982} C_VEL
LIN {X 0,Y 397.139,Z 313.512,A -85,B 0,C 180,E1 -11319.705,E2 -11319.705} C_VEL
LIN {X 0,Y 397.182,Z 313.504,A -85,B 0,C 180,E1 -11322.845,E2 -11322.845} C_VEL
LIN {X 0,Y 397.227,Z 313.494,A -85,B 0,C 180,E1 -11326.679,E2 -11326.679} C_VEL
LIN {X 0,Y 397.219,Z 313.503,A -85,B 0,C 180,E1 -11329.809,E2 -11329.809} C_VEL
LIN {X 0,Y 397.366,Z 313.484,A -85,B 0,C 180,E1 -11332.889,E2 -11332.889} C_VEL
LIN {X 0,Y 397.257,Z 313.493,A -85,B 0,C 180,E1 -11334.925,E2 -11334.925} C_VEL
LIN {X 0,Y 397.453,Z 313.474,A -85,B 0,C 180,E1 -11337.974,E2 -11337.974} C_VEL
LIN {X 0,Y 397.583,Z 313.455,A -85,B 0,C 180,E1 -11340,E2 -11340} C_VEL
LIN {X 0,Y 397.382,Z 313.484,A -85,B 0,C 180,E1 -11343.042,E2 -11343.042} C_VEL
LIN {X 0,Y 397.367,Z 313.49,A -85,B 0,C 180,E1 -11347.112,E2 -11347.112} C_VEL
LIN {X 0,Y 397.22,Z 313.502,A -85,B 0,C 180,E1 -11350.191,E2 -11350.191} C_VEL
LIN {X 0,Y 397.228,Z 313.501,A -85,B 0,C 180,E1 -11353.321,E2 -11353.321} C_VEL
LIN {X 0,Y 397.183,Z 313.507,A -85,B 0,C 180,E1 -11357.155,E2 -11357.155} C_VEL
LIN {X 0,Y 397.104,Z 313.518,A -85,B 0,C 180,E1 -11360.73,E2 -11360.73} C_VEL
LIN {X 0,Y 397.124,Z 313.519,A -85,B 0,C 180,E1 -11364.019,E2 -11364.019} C_VEL
LIN {X 0,Y 397.15,Z 313.502,A -85,B 0,C 180,E1 -11367.773,E2 -11367.773} C_VEL
LIN {X 0,Y 397.079,Z 313.519,A -85,B 0,C 180,E1 -11370.883,E2 -11370.883} C_VEL
LIN {X 0,Y 397.126,Z 313.512,A -85,B 0,C 180,E1 -11374.493,E2 -11374.493} C_VEL
LIN {X 0,Y 397.104,Z 313.517,A -85,B 0,C 180,E1 -11378.275,E2 -11378.275} C_VEL
LIN {X 0,Y 397.123,Z 313.608,A -85,B 0,C 180,E1 -11380.989,E2 -11380.989} C_VEL
LIN {X 0,Y 398.12,Z 318.141,A -85,B 0,C 180,E1 -11382.147,E2 -11382.147} C_VEL
LIN {X 0,Y 399.716,Z 326.757,A -85,B 0,C 180,E1 -11384.166,E2 -11384.166} C_VEL
LIN {X 0,Y 399.434,Z 334.567,A -85,B 0,C 180,E1 -11385.798,E2 -11385.798} C_VEL
LIN {X 0,Y 401.043,Z 342.268,A -85,B 0,C 180,E1 -11386.078,E2 -11386.078} C_VEL
LIN {X 0,Y 404.068,Z 359.374,A -85,B 0,C 180,E1 -11386.569,E2 -11386.569} C_VEL
LIN {X 0,Y 402.763,Z 440.526,A -85,B 0,C 180,E1 -11388.067,E2 -11388.067} C_VEL
LIN {X 0,Y 402.442,Z 450.687,A -85,B 0,C 180,E1 -11388.362,E2 -11388.362} C_VEL
LIN {X 0,Y 402.089,Z 460.42,A -85,B 0,C 180,E1 -11388.766,E2 -11388.766} C_VEL
LIN {X 0,Y 401.45,Z 471.658,A -85,B 0,C 180,E1 -11389.394,E2 -11389.394} C_VEL
LIN {X 0,Y 400.761,Z 481.937,A -85,B 0,C 180,E1 -11390.135,E2 -11390.135} C_VEL
LIN {X 0,Y 400.068,Z 490.962,A -85,B 0,C 180,E1 -11390.934,E2 -11390.934} C_VEL
LIN {X 0,Y 399.22,Z 500.49,A -85,B 0,C 180,E1 -11391.964,E2 -11391.964} C_VEL
LIN {X 0,Y 398.586,Z 507.86,A -85,B 0,C 180,E1 -11392.911,E2 -11392.911} C_VEL
LIN {X 0,Y 397.789,Z 516.909,A -85,B 0,C 180,E1 -11394.336,E2 -11394.336} C_VEL
LIN {X 0,Y 397.222,Z 523.165,A -85,B 0,C 180,E1 -11395.516,E2 -11395.516} C_VEL
LIN {X 0,Y 396.713,Z 529.575,A -85,B 0,C 180,E1 -11396.992,E2 -11396.992} C_VEL
LIN {X 0,Y 396.314,Z 534.375,A -85,B 0,C 180,E1 -11398.343,E2 -11398.343} C_VEL
LIN {X 0,Y 396.082,Z 538.101,A -85,B 0,C 180,E1 -11399.622,E2 -11399.622} C_VEL
LIN {X 0,Y 395.815,Z 541.838,A -85,B 0,C 180,E1 -11401.353,E2 -11401.353} C_VEL
LIN {X 0,Y 395.657,Z 543.866,A -85,B 0,C 180,E1 -11402.641,E2 -11402.641} C_VEL
LIN {X 0,Y 395.49,Z 545.63,A -85,B 0,C 180,E1 -11404.755,E2 -11404.755} C_VEL
LIN {X 0,Y 395.472,Z 545.971,A -85,B 0,C 180,E1 -11405.875,E2 -11405.875} C_VEL
LIN {X 0,Y 395.524,Z 545.503,A -85,B 0,C 180,E1 -11407.515,E2 -11407.515} C_VEL
LIN {X 0,Y 395.619,Z 543.961,A -85,B 0,C 180,E1 -11409.189,E2 -11409.189} C_VEL
LIN {X 0,Y 395.835,Z 541.37,A -85,B 0,C 180,E1 -11410.824,E2 -11410.824} C_VEL
LIN {X 0,Y 396.077,Z 537.682,A -85,B 0,C 180,E1 -11412.443,E2 -11412.443} C_VEL
LIN {X 0,Y 396.394,Z 532.791,A -85,B 0,C 180,E1 -11414.049,E2 -11414.049} C_VEL
LIN {X 0,Y 396.818,Z 526.554,A -85,B 0,C 180,E1 -11415.644,E2 -11415.644} C_VEL
LIN {X 0,Y 397.354,Z 520.202,A -85,B 0,C 180,E1 -11416.967,E2 -11416.967} C_VEL
LIN {X 0,Y 397.972,Z 512.534,A -85,B 0,C 180,E1 -11418.283,E2 -11418.283} C_VEL
LIN {X 0,Y 398.705,Z 504.207,A -85,B 0,C 180,E1 -11419.462,E2 -11419.462} C_VEL
LIN {X 0,Y 399.352,Z 495.591,A -85,B 0,C 180,E1 -11420.481,E2 -11420.481} C_VEL
LIN {X 0,Y 400.166,Z 485.954,A -85,B 0,C 180,E1 -11421.415,E2 -11421.415} C_VEL
LIN {X 0,Y 400.807,Z 476.18,A -85,B 0,C 180,E1 -11422.19,E2 -11422.19} C_VEL
LIN {X 0,Y 401.4,Z 465.992,A -85,B 0,C 180,E1 -11422.834,E2 -11422.834} C_VEL
LIN {X 0,Y 401.854,Z 455.455,A -85,B 0,C 180,E1 -11423.347,E2 -11423.347} C_VEL
LIN {X 0,Y 402.327,Z 444.101,A -85,B 0,C 180,E1 -11423.732,E2 -11423.732} C_VEL
LIN {X 0,Y 402.523,Z 431.365,A -85,B 0,C 180,E1 -11424.013,E2 -11424.013} C_VEL
LIN {X 0,Y 402.02,Z 425.553,A -85,B 0,C 180,E1 -11424.144,E2 -11424.144} C_VEL
LIN {X 0,Y 396.782,Z 406.846,A -85,B 0,C 180,E1 -11424.731,E2 -11424.731} C_VEL
LIN {X 0,Y 396.184,Z 401.034,A -85,B 0,C 180,E1 -11424.869,E2 -11424.869} C_VEL
LIN {X 0,Y 396.731,Z 358.88,A -85,B 0,C 180,E1 -11425.651,E2 -11425.651} C_VEL
LIN {X 0,Y 392.344,Z 335.468,A -85,B 0,C 180,E1 -11426.335,E2 -11426.335} C_VEL
LIN {X 0,Y 392.365,Z 333.681,A -85,B 0,C 180,E1 -11426.663,E2 -11426.663} C_VEL
LIN {X 0,Y 392.754,Z 328.375,A -85,B 0,C 180,E1 -11427.949,E2 -11427.949} C_VEL
LIN {X 0,Y 391.241,Z 318.496,A -85,B 0,C 180,E1 -11430.515,E2 -11430.515} C_VEL
LIN {X 0,Y 390.404,Z 314.398,A -85,B 0,C 180,E1 -11431.676,E2 -11431.676} C_VEL
LIN {X 0,Y 390.225,Z 314.376,A -85,B 0,C 180,E1 -11435.167,E2 -11435.167} C_VEL
LIN {X 0,Y 390.271,Z 314.366,A -85,B 0,C 180,E1 -11437.929,E2 -11437.929} C_VEL
LIN {X 0,Y 390.15,Z 314.381,A -85,B 0,C 180,E1 -11441.429,E2 -11441.429} C_VEL
LIN {X 0,Y 390.146,Z 314.382,A -85,B 0,C 180,E1 -11444.607,E2 -11444.607} C_VEL
LIN {X 0,Y 390.13,Z 314.39,A -85,B 0,C 180,E1 -11447.833,E2 -11447.833} C_VEL
LIN {X 0,Y 390.063,Z 314.394,A -85,B 0,C 180,E1 -11451.122,E2 -11451.122} C_VEL
LIN {X 0,Y 390.079,Z 314.391,A -85,B 0,C 180,E1 -11454.481,E2 -11454.481} C_VEL
LIN {X 0,Y 390.119,Z 314.379,A -85,B 0,C 180,E1 -11457.93,E2 -11457.93} C_VEL
LIN {X 0,Y 390.026,Z 314.401,A -85,B 0,C 180,E1 -11461.504,E2 -11461.504} C_VEL
LIN {X 0,Y 390.086,Z 314.382,A -85,B 0,C 180,E1 -11465.207,E2 -11465.207} C_VEL
LIN {X 0,Y 390.072,Z 314.391,A -85,B 0,C 180,E1 -11469.219,E2 -11469.219} C_VEL
LIN {X 0,Y 390.044,Z 314.388,A -85,B 0,C 180,E1 -11472.374,E2 -11472.374} C_VEL
LIN {X 0,Y 390.045,Z 314.395,A -85,B 0,C 180,E1 -11475.354,E2 -11475.354} C_VEL
LIN {X 0,Y 390.026,Z 314.396,A -85,B 0,C 180,E1 -11478.186,E2 -11478.186} C_VEL
LIN {X 0,Y 390.068,Z 314.378,A -85,B 0,C 180,E1 -11480.905,E2 -11480.905} C_VEL
LIN {X 0,Y 390.086,Z 314.39,A -85,B 0,C 180,E1 -11484.793,E2 -11484.793} C_VEL
LIN {X 0,Y 390.025,Z 314.387,A -85,B 0,C 180,E1 -11488.496,E2 -11488.496} C_VEL
LIN {X 0,Y 390.04,Z 314.383,A -85,B 0,C 180,E1 -11492.064,E2 -11492.064} C_VEL
LIN {X 0,Y 390.065,Z 314.392,A -85,B 0,C 180,E1 -11495.518,E2 -11495.518} C_VEL
LIN {X 0,Y 390.058,Z 314.387,A -85,B 0,C 180,E1 -11498.878,E2 -11498.878} C_VEL
LIN {X 0,Y 390.113,Z 314.36,A -85,B 0,C 180,E1 -11502.166,E2 -11502.166} C_VEL
LIN {X 0,Y 390.145,Z 314.384,A -85,B 0,C 180,E1 -11505.392,E2 -11505.392} C_VEL
LIN {X 0,Y 390.147,Z 314.381,A -85,B 0,C 180,E1 -11508.571,E2 -11508.571} C_VEL
LIN {X 0,Y 390.259,Z 314.35,A -85,B 0,C 180,E1 -11512.086,E2 -11512.086} C_VEL
LIN {X 0,Y 390.208,Z 314.357,A -85,B 0,C 180,E1 -11514.833,E2 -11514.833} C_VEL
LIN {X 0,Y 390.41,Z 314.348,A -85,B 0,C 180,E1 -11517.936,E2 -11517.936} C_VEL
LIN {X 0,Y 390.335,Z 314.355,A -85,B 0,C 180,E1 -11521.031,E2 -11521.031} C_VEL
LIN {X 0,Y 390.26,Z 314.354,A -85,B 0,C 180,E1 -11523.097,E2 -11523.097} C_VEL
LIN {X 0,Y 390.305,Z 314.347,A -85,B 0,C 180,E1 -11526.202,E2 -11526.202} C_VEL
LIN {X 0,Y 390.193,Z 314.383,A -85,B 0,C 180,E1 -11529.329,E2 -11529.329} C_VEL
LIN {X 0,Y 390.172,Z 314.374,A -85,B 0,C 180,E1 -11532.483,E2 -11532.483} C_VEL
LIN {X 0,Y 390.066,Z 314.378,A -85,B 0,C 180,E1 -11535.68,E2 -11535.68} C_VEL
LIN {X 0,Y 390.074,Z 314.391,A -85,B 0,C 180,E1 -11538.923,E2 -11538.923} C_VEL
LIN {X 0,Y 390.036,Z 314.394,A -85,B 0,C 180,E1 -11542.234,E2 -11542.234} C_VEL
LIN {X 0,Y 390.05,Z 314.389,A -85,B 0,C 180,E1 -11545.722,E2 -11545.722} C_VEL
LIN {X 0,Y 390.025,Z 314.398,A -85,B 0,C 180,E1 -11549.112,E2 -11549.112} C_VEL
LIN {X 0,Y 390.041,Z 314.392,A -85,B 0,C 180,E1 -11552.721,E2 -11552.721} C_VEL
LIN {X 0,Y 390.052,Z 314.394,A -85,B 0,C 180,E1 -11555.824,E2 -11555.824} C_VEL
LIN {X 0,Y 390.035,Z 314.396,A -85,B 0,C 180,E1 -11559.212,E2 -11559.212} C_VEL
LIN {X 0,Y 390.028,Z 314.396,A -85,B 0,C 180,E1 -11562.371,E2 -11562.371} C_VEL
LIN {X 0,Y 390.038,Z 314.396,A -85,B 0,C 180,E1 -11565.353,E2 -11565.353} C_VEL
LIN {X 0,Y 390.013,Z 314.403,A -85,B 0,C 180,E1 -11568.184,E2 -11568.184} C_VEL
LIN {X 0,Y 390.056,Z 314.4,A -85,B 0,C 180,E1 -11570.903,E2 -11570.903} C_VEL
LIN {X 0,Y 390.068,Z 314.396,A -85,B 0,C 180,E1 -11574.791,E2 -11574.791} C_VEL
LIN {X 0,Y 390.021,Z 314.401,A -85,B 0,C 180,E1 -11578.495,E2 -11578.495} C_VEL
LIN {X 0,Y 390.036,Z 314.401,A -85,B 0,C 180,E1 -11582.064,E2 -11582.064} C_VEL
LIN {X 0,Y 390.106,Z 314.617,A -85,B 0,C 180,E1 -11582.433,E2 -11582.433} C_VEL
LIN {X 0,Y 392.443,Z 326.369,A -85,B 0,C 180,E1 -11585.394,E2 -11585.394} C_VEL
LIN {X 0,Y 393.165,Z 331.263,A -85,B 0,C 180,E1 -11586.578,E2 -11586.578} C_VEL
LIN {X 0,Y 392.094,Z 345.239,A -85,B 0,C 180,E1 -11589.671,E2 -11589.671} C_VEL
LIN {X 0,Y 396.491,Z 371.728,A -85,B 0,C 180,E1 -11590.426,E2 -11590.426} C_VEL
LIN {X 0,Y 395.69,Z 445.361,A -85,B 0,C 180,E1 -11591.791,E2 -11591.791} C_VEL
LIN {X 0,Y 395.3,Z 460.102,A -85,B 0,C 180,E1 -11592.174,E2 -11592.174} C_VEL
LIN {X 0,Y 394.622,Z 471.542,A -85,B 0,C 180,E1 -11592.644,E2 -11592.644} C_VEL
LIN {X 0,Y 394.195,Z 480.847,A -85,B 0,C 180,E1 -11593.159,E2 -11593.159} C_VEL
LIN {X 0,Y 393.376,Z 491.641,A -85,B 0,C 180,E1 -11593.923,E2 -11593.923} C_VEL
LIN {X 0,Y 392.61,Z 502.094,A -85,B 0,C 180,E1 -11594.863,E2 -11594.863} C_VEL
LIN {X 0,Y 391.881,Z 510.917,A -85,B 0,C 180,E1 -11595.827,E2 -11595.827} C_VEL
LIN {X 0,Y 391.158,Z 519.902,A -85,B 0,C 180,E1 -11597.021,E2 -11597.021} C_VEL
LIN {X 0,Y 390.545,Z 526.524,A -85,B 0,C 180,E1 -11598.056,E2 -11598.056} C_VEL
LIN {X 0,Y 389.937,Z 533.466,A -85,B 0,C 180,E1 -11599.354,E2 -11599.354} C_VEL
LIN {X 0,Y 389.46,Z 539.27,A -85,B 0,C 180,E1 -11600.653,E2 -11600.653} C_VEL
LIN {X 0,Y 389.086,Z 544.889,A -85,B 0,C 180,E1 -11602.214,E2 -11602.214} C_VEL
LIN {X 0,Y 388.83,Z 549.313,A -85,B 0,C 180,E1 -11603.774,E2 -11603.774} C_VEL
LIN {X 0,Y 388.757,Z 551.63,A -85,B 0,C 180,E1 -11604.814,E2 -11604.814} C_VEL
LIN {X 0,Y 388.597,Z 555.025,A -85,B 0,C 180,E1 -11606.89,E2 -11606.89} C_VEL
LIN {X 0,Y 388.649,Z 556.625,A -85,B 0,C 180,E1 -11608.964,E2 -11608.964} C_VEL
LIN {X 0,Y 388.667,Z 556.938,A -85,B 0,C 180,E1 -11610,E2 -11610} C_VEL
LIN {X 0,Y 388.611,Z 556.155,A -85,B 0,C 180,E1 -11612.073,E2 -11612.073} C_VEL
LIN {X 0,Y 388.597,Z 555.181,A -85,B 0,C 180,E1 -11613.11,E2 -11613.11} C_VEL
LIN {X 0,Y 388.797,Z 552.024,A -85,B 0,C 180,E1 -11615.185,E2 -11615.185} C_VEL
LIN {X 0,Y 388.909,Z 548.466,A -85,B 0,C 180,E1 -11616.746,E2 -11616.746} C_VEL
LIN {X 0,Y 389.215,Z 543.799,A -85,B 0,C 180,E1 -11618.306,E2 -11618.306} C_VEL
LIN {X 0,Y 389.684,Z 537.871,A -85,B 0,C 180,E1 -11619.865,E2 -11619.865} C_VEL
LIN {X 0,Y 390.289,Z 530.461,A -85,B 0,C 180,E1 -11621.425,E2 -11621.425} C_VEL
LIN {X 0,Y 391.078,Z 522.957,A -85,B 0,C 180,E1 -11622.717,E2 -11622.717} C_VEL
LIN {X 0,Y 391.758,Z 515.942,A -85,B 0,C 180,E1 -11623.743,E2 -11623.743} C_VEL
LIN {X 0,Y 392.488,Z 506.878,A -85,B 0,C 180,E1 -11624.849,E2 -11624.849} C_VEL
LIN {X 0,Y 393.295,Z 497.237,A -85,B 0,C 180,E1 -11625.814,E2 -11625.814} C_VEL
LIN {X 0,Y 394.071,Z 487.885,A -85,B 0,C 180,E1 -11626.58,E2 -11626.58} C_VEL
LIN {X 0,Y 394.847,Z 477.091,A -85,B 0,C 180,E1 -11627.279,E2 -11627.279} C_VEL
LIN {X 0,Y 395.483,Z 465.334,A -85,B 0,C 180,E1 -11627.851,E2 -11627.851} C_VEL
LIN {X 0,Y 395.959,Z 455.433,A -85,B 0,C 180,E1 -11628.196,E2 -11628.196} C_VEL
LIN {X 0,Y 396.301,Z 439.26,A -85,B 0,C 180,E1 -11628.548,E2 -11628.548} C_VEL
LIN {X 0,Y 397.092,Z 371.704,A -85,B 0,C 180,E1 -11629.812,E2 -11629.812} C_VEL
LIN {X 0,Y 392.617,Z 346.314,A -85,B 0,C 180,E1 -11630.566,E2 -11630.566} C_VEL
LIN {X 0,Y 392.357,Z 344.718,A -85,B 0,C 180,E1 -11630.652,E2 -11630.652} C_VEL
LIN {X 0,Y 393.309,Z 331.935,A -85,B 0,C 180,E1 -11633.421,E2 -11633.421} C_VEL
LIN {X 0,Y 392.667,Z 326.98,A -85,B 0,C 180,E1 -11634.591,E2 -11634.591} C_VEL
LIN {X 0,Y 390.369,Z 315.898,A -85,B 0,C 180,E1 -11637.328,E2 -11637.328} C_VEL
LIN {X 0,Y 390.063,Z 314.429,A -85,B 0,C 180,E1 -11637.788,E2 -11637.788} C_VEL
LIN {X 0,Y 390.021,Z 314.4,A -85,B 0,C 180,E1 -11641.505,E2 -11641.505} C_VEL
LIN {X 0,Y 390.082,Z 314.395,A -85,B 0,C 180,E1 -11645.207,E2 -11645.207} C_VEL
LIN {X 0,Y 390.085,Z 314.391,A -85,B 0,C 180,E1 -11649.093,E2 -11649.093} C_VEL
LIN {X 0,Y 390.037,Z 314.399,A -85,B 0,C 180,E1 -11652.374,E2 -11652.374} C_VEL
LIN {X 0,Y 390.043,Z 314.399,A -85,B 0,C 180,E1 -11655.355,E2 -11655.355} C_VEL
LIN {X 0,Y 390.029,Z 314.395,A -85,B 0,C 180,E1 -11658.187,E2 -11658.187} C_VEL
LIN {X 0,Y 390.086,Z 314.391,A -85,B 0,C 180,E1 -11660.908,E2 -11660.908} C_VEL
LIN {X 0,Y 390.084,Z 314.386,A -85,B 0,C 180,E1 -11664.793,E2 -11664.793} C_VEL
LIN {X 0,Y 390.023,Z 314.398,A -85,B 0,C 180,E1 -11668.496,E2 -11668.496} C_VEL
LIN {X 0,Y 390.117,Z 314.388,A -85,B 0,C 180,E1 -11672.07,E2 -11672.07} C_VEL
LIN {X 0,Y 390.08,Z 314.39,A -85,B 0,C 180,E1 -11675.52,E2 -11675.52} C_VEL
LIN {X 0,Y 390.056,Z 314.398,A -85,B 0,C 180,E1 -11678.878,E2 -11678.878} C_VEL
LIN {X 0,Y 390.129,Z 314.381,A -85,B 0,C 180,E1 -11682.167,E2 -11682.167} C_VEL
LIN {X 0,Y 390.145,Z 314.383,A -85,B 0,C 180,E1 -11685.393,E2 -11685.393} C_VEL
LIN {X 0,Y 390.149,Z 314.383,A -85,B 0,C 180,E1 -11688.572,E2 -11688.572} C_VEL
LIN {X 0,Y 390.345,Z 314.357,A -85,B 0,C 180,E1 -11691.993,E2 -11691.993} C_VEL
LIN {X 0,Y 390.229,Z 314.369,A -85,B 0,C 180,E1 -11694.834,E2 -11694.834} C_VEL
LIN {X 0,Y 390.422,Z 314.35,A -85,B 0,C 180,E1 -11697.937,E2 -11697.937} C_VEL
LIN {X 0,Y 390.552,Z 314.331,A -85,B 0,C 180,E1 -11700,E2 -11700} C_VEL
LIN {X 0,Y 390.316,Z 314.364,A -85,B 0,C 180,E1 -11703.097,E2 -11703.097} C_VEL
LIN {X 0,Y 390.313,Z 314.361,A -85,B 0,C 180,E1 -11706.62,E2 -11706.62} C_VEL
LIN {X 0,Y 390.207,Z 314.376,A -85,B 0,C 180,E1 -11709.329,E2 -11709.329} C_VEL
LIN {X 0,Y 390.173,Z 314.375,A -85,B 0,C 180,E1 -11712.483,E2 -11712.483} C_VEL
LIN {X 0,Y 390.141,Z 314.386,A -85,B 0,C 180,E1 -11715.677,E2 -11715.677} C_VEL
LIN {X 0,Y 390.107,Z 314.385,A -85,B 0,C 180,E1 -11718.922,E2 -11718.922} C_VEL
LIN {X 0,Y 390.039,Z 314.4,A -85,B 0,C 180,E1 -11722.234,E2 -11722.234} C_VEL
LIN {X 0,Y 390.085,Z 314.393,A -85,B 0,C 180,E1 -11725.733,E2 -11725.733} C_VEL
LIN {X 0,Y 390.09,Z 314.382,A -85,B 0,C 180,E1 -11728.018,E2 -11728.018} C_VEL
LIN {X 0,Y 390.024,Z 314.397,A -85,B 0,C 180,E1 -11731.505,E2 -11731.505} C_VEL
LIN {X 0,Y 390.085,Z 314.397,A -85,B 0,C 180,E1 -11735.207,E2 -11735.207} C_VEL
LIN {X 0,Y 390.071,Z 314.399,A -85,B 0,C 180,E1 -11739.219,E2 -11739.219} C_VEL
LIN {X 0,Y 390.13,Z 314.622,A -85,B 0,C 180,E1 -11740.735,E2 -11740.735} C_VEL
LIN {X 0,Y 392.531,Z 326.199,A -85,B 0,C 180,E1 -11743.576,E2 -11743.576} C_VEL
LIN {X 0,Y 392.737,Z 331.18,A -85,B 0,C 180,E1 -11744.705,E2 -11744.705} C_VEL
LIN {X 0,Y 392.601,Z 334.739,A -85,B 0,C 180,E1 -11745.415,E2 -11745.415} C_VEL
LIN {X 0,Y 396.294,Z 353.038,A -85,B 0,C 180,E1 -11746.024,E2 -11746.024} C_VEL
LIN {X 0,Y 397.415,Z 359.776,A -85,B 0,C 180,E1 -11746.218,E2 -11746.218} C_VEL
LIN {X 0,Y 396.072,Z 440.699,A -85,B 0,C 180,E1 -11747.739,E2 -11747.739} C_VEL
LIN {X 0,Y 395.739,Z 450.473,A -85,B 0,C 180,E1 -11748.023,E2 -11748.023} C_VEL
LIN {X 0,Y 395.379,Z 460.238,A -85,B 0,C 180,E1 -11748.432,E2 -11748.432} C_VEL
LIN {X 0,Y 394.728,Z 471.217,A -85,B 0,C 180,E1 -11749.048,E2 -11749.048} C_VEL
LIN {X 0,Y 394.075,Z 480.699,A -85,B 0,C 180,E1 -11749.723,E2 -11749.723} C_VEL
LIN {X 0,Y 393.263,Z 490.811,A -85,B 0,C 180,E1 -11750.623,E2 -11750.623} C_VEL
LIN {X 0,Y 392.366,Z 500.528,A -85,B 0,C 180,E1 -11751.689,E2 -11751.689} C_VEL
LIN {X 0,Y 391.626,Z 508.384,A -85,B 0,C 180,E1 -11752.723,E2 -11752.723} C_VEL
LIN {X 0,Y 390.903,Z 516.434,A -85,B 0,C 180,E1 -11754.003,E2 -11754.003} C_VEL
LIN {X 0,Y 390.193,Z 523.826,A -85,B 0,C 180,E1 -11755.434,E2 -11755.434} C_VEL
LIN {X 0,Y 389.766,Z 529.029,A -85,B 0,C 180,E1 -11756.636,E2 -11756.636} C_VEL
LIN {X 0,Y 389.327,Z 534.048,A -85,B 0,C 180,E1 -11758.041,E2 -11758.041} C_VEL
LIN {X 0,Y 389.005,Z 538.473,A -85,B 0,C 180,E1 -11759.611,E2 -11759.611} C_VEL
LIN {X 0,Y 388.82,Z 541.08,A -85,B 0,C 180,E1 -11760.789,E2 -11760.789} C_VEL
LIN {X 0,Y 388.575,Z 543.728,A -85,B 0,C 180,E1 -11762.405,E2 -11762.405} C_VEL
LIN {X 0,Y 388.413,Z 545.559,A -85,B 0,C 180,E1 -11764.262,E2 -11764.262} C_VEL
LIN {X 0,Y 388.388,Z 545.938,A -85,B 0,C 180,E1 -11765.406,E2 -11765.406} C_VEL
LIN {X 0,Y 388.435,Z 545.521,A -85,B 0,C 180,E1 -11767.669,E2 -11767.669} C_VEL
LIN {X 0,Y 388.486,Z 544.489,A -85,B 0,C 180,E1 -11768.788,E2 -11768.788} C_VEL
LIN {X 0,Y 388.768,Z 541.244,A -85,B 0,C 180,E1 -11771.01,E2 -11771.01} C_VEL
LIN {X 0,Y 389.032,Z 537.305,A -85,B 0,C 180,E1 -11772.712,E2 -11772.712} C_VEL
LIN {X 0,Y 389.374,Z 532.477,A -85,B 0,C 180,E1 -11774.292,E2 -11774.292} C_VEL
LIN {X 0,Y 389.751,Z 527.366,A -85,B 0,C 180,E1 -11775.644,E2 -11775.644} C_VEL
LIN {X 0,Y 390.299,Z 520.848,A -85,B 0,C 180,E1 -11777.049,E2 -11777.049} C_VEL
LIN {X 0,Y 390.915,Z 513.658,A -85,B 0,C 180,E1 -11778.331,E2 -11778.331} C_VEL
LIN {X 0,Y 391.747,Z 504.474,A -85,B 0,C 180,E1 -11779.665,E2 -11779.665} C_VEL
LIN {X 0,Y 392.438,Z 495.665,A -85,B 0,C 180,E1 -11780.725,E2 -11780.725} C_VEL
LIN {X 0,Y 393.284,Z 486.273,A -85,B 0,C 180,E1 -11781.652,E2 -11781.652} C_VEL
LIN {X 0,Y 393.949,Z 476.547,A -85,B 0,C 180,E1 -11782.44,E2 -11782.44} C_VEL
LIN {X 0,Y 394.543,Z 466.453,A -85,B 0,C 180,E1 -11783.094,E2 -11783.094} C_VEL
LIN {X 0,Y 395.079,Z 455.151,A -85,B 0,C 180,E1 -11783.649,E2 -11783.649} C_VEL
LIN {X 0,Y 395.541,Z 444.567,A -85,B 0,C 180,E1 -11784.016,E2 -11784.016} C_VEL
LIN {X 0,Y 395.795,Z 428.511,A -85,B 0,C 180,E1 -11784.365,E2 -11784.365} C_VEL
LIN {X 0,Y 396.184,Z 401.034,A -85,B 0,C 180,E1 -11784.869,E2 -11784.869} C_VEL
LIN {X 0,Y 395.6,Z 395.225,A -85,B 0,C 180,E1 -11785.008,E2 -11785.008} C_VEL
LIN {X 0,Y 390.462,Z 376.517,A -85,B 0,C 180,E1 -11785.617,E2 -11785.617} C_VEL
LIN {X 0,Y 389.951,Z 370.707,A -85,B 0,C 180,E1 -11785.756,E2 -11785.756} C_VEL
LIN {X 0,Y 389.927,Z 359.203,A -85,B 0,C 180,E1 -11785.983,E2 -11785.983} C_VEL
LIN {X 0,Y 385.431,Z 335.242,A -85,B 0,C 180,E1 -11786.717,E2 -11786.717} C_VEL
LIN {X 0,Y 385.754,Z 329.148,A -85,B 0,C 180,E1 -11788.173,E2 -11788.173} C_VEL
LIN {X 0,Y 384.383,Z 320.264,A -85,B 0,C 180,E1 -11790.524,E2 -11790.524} C_VEL
LIN {X 0,Y 383.389,Z 315.285,A -85,B 0,C 180,E1 -11791.937,E2 -11791.937} C_VEL
LIN {X 0,Y 383.274,Z 315.238,A -85,B 0,C 180,E1 -11796.317,E2 -11796.317} C_VEL
LIN {X 0,Y 383.145,Z 315.26,A -85,B 0,C 180,E1 -11799.502,E2 -11799.502} C_VEL
LIN {X 0,Y 383.127,Z 315.261,A -85,B 0,C 180,E1 -11803.536,E2 -11803.536} C_VEL
LIN {X 0,Y 383.097,Z 315.263,A -85,B 0,C 180,E1 -11807.455,E2 -11807.455} C_VEL
LIN {X 0,Y 383.036,Z 315.273,A -85,B 0,C 180,E1 -11810.649,E2 -11810.649} C_VEL
LIN {X 0,Y 383.027,Z 315.264,A -85,B 0,C 180,E1 -11813.808,E2 -11813.808} C_VEL
LIN {X 0,Y 383.081,Z 315.264,A -85,B 0,C 180,E1 -11816.123,E2 -11816.123} C_VEL
LIN {X 0,Y 382.994,Z 315.274,A -85,B 0,C 180,E1 -11819.7,E2 -11819.7} C_VEL
LIN {X 0,Y 383.005,Z 315.268,A -85,B 0,C 180,E1 -11823.401,E2 -11823.401} C_VEL
LIN {X 0,Y 383.033,Z 315.27,A -85,B 0,C 180,E1 -11826.165,E2 -11826.165} C_VEL
LIN {X 0,Y 383.011,Z 315.27,A -85,B 0,C 180,E1 -11829.958,E2 -11829.958} C_VEL
LIN {X 0,Y 383.007,Z 315.267,A -85,B 0,C 180,E1 -11832.779,E2 -11832.779} C_VEL
LIN {X 0,Y 382.998,Z 315.273,A -85,B 0,C 180,E1 -11835.789,E2 -11835.789} C_VEL
LIN {X 0,Y 382.972,Z 315.268,A -85,B 0,C 180,E1 -11838.799,E2 -11838.799} C_VEL
LIN {X 0,Y 382.998,Z 315.262,A -85,B 0,C 180,E1 -11842.097,E2 -11842.097} C_VEL
LIN {X 0,Y 383.02,Z 315.276,A -85,B 0,C 180,E1 -11845.332,E2 -11845.332} C_VEL
LIN {X 0,Y 382.984,Z 315.265,A -85,B 0,C 180,E1 -11849.081,E2 -11849.081} C_VEL
LIN {X 0,Y 382.995,Z 315.265,A -85,B 0,C 180,E1 -11852.693,E2 -11852.693} C_VEL
LIN {X 0,Y 383.024,Z 315.275,A -85,B 0,C 180,E1 -11856.192,E2 -11856.192} C_VEL
LIN {X 0,Y 383.058,Z 315.254,A -85,B 0,C 180,E1 -11859.598,E2 -11859.598} C_VEL
LIN {X 0,Y 383.096,Z 315.24,A -85,B 0,C 180,E1 -11862.931,E2 -11862.931} C_VEL
LIN {X 0,Y 383.128,Z 315.254,A -85,B 0,C 180,E1 -11866.464,E2 -11866.464} C_VEL
LIN {X 0,Y 383.144,Z 315.247,A -85,B 0,C 180,E1 -11870.497,E2 -11870.497} C_VEL
LIN {X 0,Y 383.242,Z 315.22,A -85,B 0,C 180,E1 -11873.683,E2 -11873.683} C_VEL
LIN {X 0,Y 383.376,Z 315.224,A -85,B 0,C 180,E1 -11877.899,E2 -11877.899} C_VEL
LIN {X 0,Y 383.302,Z 315.231,A -85,B 0,C 180,E1 -11881.05,E2 -11881.05} C_VEL
LIN {X 0,Y 383.198,Z 315.233,A -85,B 0,C 180,E1 -11883.154,E2 -11883.154} C_VEL
LIN {X 0,Y 383.262,Z 315.224,A -85,B 0,C 180,E1 -11886.316,E2 -11886.316} C_VEL
LIN {X 0,Y 383.143,Z 315.259,A -85,B 0,C 180,E1 -11889.502,E2 -11889.502} C_VEL
LIN {X 0,Y 383.127,Z 315.248,A -85,B 0,C 180,E1 -11893.536,E2 -11893.536} C_VEL
LIN {X 0,Y 383.053,Z 315.26,A -85,B 0,C 180,E1 -11897.434,E2 -11897.434} C_VEL
LIN {X 0,Y 383.03,Z 315.27,A -85,B 0,C 180,E1 -11900.646,E2 -11900.646} C_VEL
LIN {X 0,Y 383.01,Z 315.258,A -85,B 0,C 180,E1 -11903.808,E2 -11903.808} C_VEL
LIN {X 0,Y 382.971,Z 315.278,A -85,B 0,C 180,E1 -11907.308,E2 -11907.308} C_VEL
LIN {X 0,Y 382.981,Z 315.27,A -85,B 0,C 180,E1 -11910.918,E2 -11910.918} C_VEL
LIN {X 0,Y 383.016,Z 315.272,A -85,B 0,C 180,E1 -11914.668,E2 -11914.668} C_VEL
LIN {X 0,Y 382.992,Z 315.272,A -85,B 0,C 180,E1 -11917.902,E2 -11917.902} C_VEL
LIN {X 0,Y 382.959,Z 315.278,A -85,B 0,C 180,E1 -11921.35,E2 -11921.35} C_VEL
LIN {X 0,Y 382.987,Z 315.28,A -85,B 0,C 180,E1 -11924.302,E2 -11924.302} C_VEL
LIN {X 0,Y 382.98,Z 315.277,A -85,B 0,C 180,E1 -11927.236,E2 -11927.236} C_VEL
LIN {X 0,Y 382.984,Z 315.278,A -85,B 0,C 180,E1 -11930.419,E2 -11930.419} C_VEL
LIN {X 0,Y 383.013,Z 315.272,A -85,B 0,C 180,E1 -11934.043,E2 -11934.043} C_VEL
LIN {X 0,Y 382.984,Z 315.28,A -85,B 0,C 180,E1 -11937.578,E2 -11937.578} C_VEL
LIN {X 0,Y 382.979,Z 315.282,A -85,B 0,C 180,E1 -11940.299,E2 -11940.299} C_VEL
LIN {X 0,Y 383.015,Z 315.43,A -85,B 0,C 180,E1 -11942.118,E2 -11942.118} C_VEL
LIN {X 0,Y 385.218,Z 326.179,A -85,B 0,C 180,E1 -11944.901,E2 -11944.901} C_VEL
LIN {X 0,Y 386.222,Z 332.236,A -85,B 0,C 180,E1 -11946.401,E2 -11946.401} C_VEL
LIN {X 0,Y 385.21,Z 345.01,A -85,B 0,C 180,E1 -11949.299,E2 -11949.299} C_VEL
LIN {X 0,Y 387.255,Z 357.025,A -85,B 0,C 180,E1 -11949.681,E2 -11949.681} C_VEL
LIN {X 0,Y 389.876,Z 373.356,A -85,B 0,C 180,E1 -11950.132,E2 -11950.132} C_VEL
LIN {X 0,Y 388.77,Z 451.41,A -85,B 0,C 180,E1 -11951.625,E2 -11951.625} C_VEL
LIN {X 0,Y 388.459,Z 461.146,A -85,B 0,C 180,E1 -11951.917,E2 -11951.917} C_VEL
LIN {X 0,Y 387.834,Z 471.065,A -85,B 0,C 180,E1 -11952.33,E2 -11952.33} C_VEL
LIN {X 0,Y 387.239,Z 482.328,A -85,B 0,C 180,E1 -11952.983,E2 -11952.983} C_VEL
LIN {X 0,Y 386.41,Z 492.812,A -85,B 0,C 180,E1 -11953.761,E2 -11953.761} C_VEL
LIN {X 0,Y 385.781,Z 501.432,A -85,B 0,C 180,E1 -11954.548,E2 -11954.548} C_VEL
LIN {X 0,Y 384.913,Z 511.243,A -85,B 0,C 180,E1 -11955.642,E2 -11955.642} C_VEL
LIN {X 0,Y 384.208,Z 519.67,A -85,B 0,C 180,E1 -11956.782,E2 -11956.782} C_VEL
LIN {X 0,Y 383.585,Z 526.316,A -85,B 0,C 180,E1 -11957.836,E2 -11957.836} C_VEL
LIN {X 0,Y 382.92,Z 533.276,A -85,B 0,C 180,E1 -11959.156,E2 -11959.156} C_VEL
LIN {X 0,Y 382.428,Z 539.096,A -85,B 0,C 180,E1 -11960.48,E2 -11960.48} C_VEL
LIN {X 0,Y 382.043,Z 544.735,A -85,B 0,C 180,E1 -11962.07,E2 -11962.07} C_VEL
LIN {X 0,Y 381.731,Z 549.517,A -85,B 0,C 180,E1 -11963.815,E2 -11963.815} C_VEL
LIN {X 0,Y 381.662,Z 551.492,A -85,B 0,C 180,E1 -11964.717,E2 -11964.717} C_VEL
LIN {X 0,Y 381.511,Z 554.908,A -85,B 0,C 180,E1 -11966.832,E2 -11966.832} C_VEL
LIN {X 0,Y 381.548,Z 556.52,A -85,B 0,C 180,E1 -11968.944,E2 -11968.944} C_VEL
LIN {X 0,Y 381.567,Z 556.836,A -85,B 0,C 180,E1 -11970,E2 -11970} C_VEL
LIN {X 0,Y 381.509,Z 556.071,A -85,B 0,C 180,E1 -11972.111,E2 -11972.111} C_VEL
LIN {X 0,Y 381.512,Z 555.097,A -85,B 0,C 180,E1 -11973.168,E2 -11973.168} C_VEL
LIN {X 0,Y 381.696,Z 551.96,A -85,B 0,C 180,E1 -11975.282,E2 -11975.282} C_VEL
LIN {X 0,Y 381.845,Z 548.411,A -85,B 0,C 180,E1 -11976.871,E2 -11976.871} C_VEL
LIN {X 0,Y 382.163,Z 543.757,A -85,B 0,C 180,E1 -11978.46,E2 -11978.46} C_VEL
LIN {X 0,Y 382.68,Z 537.843,A -85,B 0,C 180,E1 -11980.048,E2 -11980.048} C_VEL
LIN {X 0,Y 383.312,Z 530.447,A -85,B 0,C 180,E1 -11981.635,E2 -11981.635} C_VEL
LIN {X 0,Y 384.128,Z 522.958,A -85,B 0,C 180,E1 -11982.951,E2 -11982.951} C_VEL
LIN {X 0,Y 384.827,Z 516.133,A -85,B 0,C 180,E1 -11983.973,E2 -11983.973} C_VEL
LIN {X 0,Y 385.655,Z 506.673,A -85,B 0,C 180,E1 -11985.146,E2 -11985.146} C_VEL
LIN {X 0,Y 386.479,Z 497.312,A -85,B 0,C 180,E1 -11986.1,E2 -11986.1} C_VEL
LIN {X 0,Y 387.289,Z 488.003,A -85,B 0,C 180,E1 -11986.879,E2 -11986.879} C_VEL
LIN {X 0,Y 388.079,Z 477.274,A -85,B 0,C 180,E1 -11987.59,E2 -11987.59} C_VEL
LIN {X 0,Y 388.752,Z 465.634,A -85,B 0,C 180,E1 -11988.171,E2 -11988.171} C_VEL
LIN {X 0,Y 389.284,Z 454.696,A -85,B 0,C 180,E1 -11988.554,E2 -11988.554} C_VEL
LIN {X 0,Y 389.676,Z 436.613,A -85,B 0,C 180,E1 -11988.944,E2 -11988.944} C_VEL
LIN {X 0,Y 390.479,Z 372.652,A -85,B 0,C 180,E1 -11990.163,E2 -11990.163} C_VEL
LIN {X 0,Y 385.874,Z 346.721,A -85,B 0,C 180,E1 -11990.956,E2 -11990.956} C_VEL
LIN {X 0,Y 385.513,Z 344.533,A -85,B 0,C 180,E1 -11991.075,E2 -11991.075} C_VEL
LIN {X 0,Y 386.418,Z 333.139,A -85,B 0,C 180,E1 -11993.586,E2 -11993.586} C_VEL
LIN {X 0,Y 384.981,Z 324.511,A -85,B 0,C 180,E1 -11995.694,E2 -11995.694} C_VEL
LIN {X 0,Y 383.007,Z 315.38,A -85,B 0,C 180,E1 -11998.085,E2 -11998.085} C_VEL
LIN {X 0,Y 382.98,Z 315.28,A -85,B 0,C 180,E1 -12000.919,E2 -12000.919} C_VEL
LIN {X 0,Y 383.016,Z 315.274,A -85,B 0,C 180,E1 -12004.668,E2 -12004.668} C_VEL
LIN {X 0,Y 382.996,Z 315.275,A -85,B 0,C 180,E1 -12007.904,E2 -12007.904} C_VEL
LIN {X 0,Y 382.968,Z 315.279,A -85,B 0,C 180,E1 -12011.349,E2 -12011.349} C_VEL
LIN {X 0,Y 382.994,Z 315.275,A -85,B 0,C 180,E1 -12014.304,E2 -12014.304} C_VEL
LIN {X 0,Y 383.009,Z 315.277,A -85,B 0,C 180,E1 -12017.24,E2 -12017.24} C_VEL
LIN {X 0,Y 383.012,Z 315.272,A -85,B 0,C 180,E1 -12020.414,E2 -12020.414} C_VEL
LIN {X 0,Y 383.024,Z 315.272,A -85,B 0,C 180,E1 -12024.045,E2 -12024.045} C_VEL
LIN {X 0,Y 382.986,Z 315.276,A -85,B 0,C 180,E1 -12027.578,E2 -12027.578} C_VEL
LIN {X 0,Y 382.992,Z 315.278,A -85,B 0,C 180,E1 -12030.301,E2 -12030.301} C_VEL
LIN {X 0,Y 383.08,Z 315.262,A -85,B 0,C 180,E1 -12034.021,E2 -12034.021} C_VEL
LIN {X 0,Y 383.009,Z 315.271,A -85,B 0,C 180,E1 -12037.336,E2 -12037.336} C_VEL
LIN {X 0,Y 383.061,Z 315.267,A -85,B 0,C 180,E1 -12040.717,E2 -12040.717} C_VEL
LIN {X 0,Y 383.082,Z 315.264,A -85,B 0,C 180,E1 -12044.027,E2 -12044.027} C_VEL
LIN {X 0,Y 383.137,Z 315.252,A -85,B 0,C 180,E1 -12047.284,E2 -12047.284} C_VEL
LIN {X 0,Y 383.153,Z 315.247,A -85,B 0,C 180,E1 -12050.498,E2 -12050.498} C_VEL
LIN {X 0,Y 383.275,Z 315.24,A -85,B 0,C 180,E1 -12052.626,E2 -12052.626} C_VEL
LIN {X 0,Y 383.201,Z 315.245,A -85,B 0,C 180,E1 -12054.739,E2 -12054.739} C_VEL
LIN {X 0,Y 383.389,Z 315.226,A -85,B 0,C 180,E1 -12057.899,E2 -12057.899} C_VEL
LIN {X 0,Y 383.521,Z 315.207,A -85,B 0,C 180,E1 -12060,E2 -12060} C_VEL
LIN {X 0,Y 383.252,Z 315.243,A -85,B 0,C 180,E1 -12063.154,E2 -12063.154} C_VEL
LIN {X 0,Y 383.273,Z 315.238,A -85,B 0,C 180,E1 -12066.614,E2 -12066.614} C_VEL
LIN {X 0,Y 383.261,Z 315.239,A -85,B 0,C 180,E1 -12068.436,E2 -12068.436} C_VEL
LIN {X 0,Y 383.1,Z 315.261,A -85,B 0,C 180,E1 -12071.642,E2 -12071.642} C_VEL
LIN {X 0,Y 383.112,Z 315.261,A -85,B 0,C 180,E1 -12074.882,E2 -12074.882} C_VEL
LIN {X 0,Y 383.064,Z 315.267,A -85,B 0,C 180,E1 -12078.174,E2 -12078.174} C_VEL
LIN {X 0,Y 382.993,Z 315.276,A -85,B 0,C 180,E1 -12081.531,E2 -12081.531} C_VEL
LIN {X 0,Y 383.029,Z 315.273,A -85,B 0,C 180,E1 -12084.962,E2 -12084.962} C_VEL
LIN {X 0,Y 383.013,Z 315.268,A -85,B 0,C 180,E1 -12088.495,E2 -12088.495} C_VEL
LIN {X 0,Y 383.01,Z 315.273,A -85,B 0,C 180,E1 -12092.15,E2 -12092.15} C_VEL
LIN {X 0,Y 383.019,Z 315.271,A -85,B 0,C 180,E1 -12094.668,E2 -12094.668} C_VEL
LIN {X 0,Y 383.001,Z 315.275,A -85,B 0,C 180,E1 -12097.904,E2 -12097.904} C_VEL
LIN {X 0,Y 383.07,Z 315.475,A -85,B 0,C 180,E1 -12100.381,E2 -12100.381} C_VEL
LIN {X 0,Y 385.354,Z 326.486,A -85,B 0,C 180,E1 -12103.155,E2 -12103.155} C_VEL
LIN {X 0,Y 385.857,Z 329.144,A -85,B 0,C 180,E1 -12103.799,E2 -12103.799} C_VEL
LIN {X 0,Y 385.756,Z 334.638,A -85,B 0,C 180,E1 -12104.989,E2 -12104.989} C_VEL
LIN {X 0,Y 386.937,Z 340.447,A -85,B 0,C 180,E1 -12105.226,E2 -12105.226} C_VEL
LIN {X 0,Y 390.754,Z 360.304,A -85,B 0,C 180,E1 -12105.851,E2 -12105.851} C_VEL
LIN {X 0,Y 389.385,Z 440.817,A -85,B 0,C 180,E1 -12107.395,E2 -12107.395} C_VEL
LIN {X 0,Y 389.013,Z 451.029,A -85,B 0,C 180,E1 -12107.702,E2 -12107.702} C_VEL
LIN {X 0,Y 388.561,Z 461.603,A -85,B 0,C 180,E1 -12108.167,E2 -12108.167} C_VEL
LIN {X 0,Y 387.931,Z 472.042,A -85,B 0,C 180,E1 -12108.777,E2 -12108.777} C_VEL
LIN {X 0,Y 387.186,Z 482.033,A -85,B 0,C 180,E1 -12109.52,E2 -12109.52} C_VEL
LIN {X 0,Y 386.459,Z 490.936,A -85,B 0,C 180,E1 -12110.331,E2 -12110.331} C_VEL
LIN {X 0,Y 385.548,Z 500.282,A -85,B 0,C 180,E1 -12111.368,E2 -12111.368} C_VEL
LIN {X 0,Y 384.649,Z 509.299,A -85,B 0,C 180,E1 -12112.59,E2 -12112.59} C_VEL
LIN {X 0,Y 383.895,Z 517.128,A -85,B 0,C 180,E1 -12113.876,E2 -12113.876} C_VEL
LIN {X 0,Y 383.284,Z 523.122,A -85,B 0,C 180,E1 -12115.04,E2 -12115.04} C_VEL
LIN {X 0,Y 382.72,Z 529.583,A -85,B 0,C 180,E1 -12116.571,E2 -12116.571} C_VEL
LIN {X 0,Y 382.321,Z 533.885,A -85,B 0,C 180,E1 -12117.786,E2 -12117.786} C_VEL
LIN {X 0,Y 381.948,Z 538.597,A -85,B 0,C 180,E1 -12119.486,E2 -12119.486} C_VEL
LIN {X 0,Y 381.732,Z 541.444,A -85,B 0,C 180,E1 -12120.798,E2 -12120.798} C_VEL
LIN {X 0,Y 381.452,Z 544.179,A -85,B 0,C 180,E1 -12122.574,E2 -12122.574} C_VEL
LIN {X 0,Y 381.309,Z 545.799,A -85,B 0,C 180,E1 -12124.573,E2 -12124.573} C_VEL
LIN {X 0,Y 381.27,Z 546.159,A -85,B 0,C 180,E1 -12126.076,E2 -12126.076} C_VEL
LIN {X 0,Y 381.316,Z 545.803,A -85,B 0,C 180,E1 -12127.229,E2 -12127.229} C_VEL
LIN {X 0,Y 381.451,Z 543.839,A -85,B 0,C 180,E1 -12129.509,E2 -12129.509} C_VEL
LIN {X 0,Y 381.722,Z 541.082,A -85,B 0,C 180,E1 -12131.204,E2 -12131.204} C_VEL
LIN {X 0,Y 382.006,Z 536.666,A -85,B 0,C 180,E1 -12133.073,E2 -12133.073} C_VEL
LIN {X 0,Y 382.343,Z 532.152,A -85,B 0,C 180,E1 -12134.542,E2 -12134.542} C_VEL
LIN {X 0,Y 382.757,Z 526.944,A -85,B 0,C 180,E1 -12135.919,E2 -12135.919} C_VEL
LIN {X 0,Y 383.33,Z 520.632,A -85,B 0,C 180,E1 -12137.291,E2 -12137.291} C_VEL
LIN {X 0,Y 384.014,Z 512.999,A -85,B 0,C 180,E1 -12138.654,E2 -12138.654} C_VEL
LIN {X 0,Y 384.863,Z 504.101,A -85,B 0,C 180,E1 -12139.955,E2 -12139.955} C_VEL
LIN {X 0,Y 385.539,Z 495.929,A -85,B 0,C 180,E1 -12140.954,E2 -12140.954} C_VEL
LIN {X 0,Y 386.407,Z 486.577,A -85,B 0,C 180,E1 -12141.897,E2 -12141.897} C_VEL
LIN {X 0,Y 387.106,Z 476.892,A -85,B 0,C 180,E1 -12142.699,E2 -12142.699} C_VEL
LIN {X 0,Y 387.724,Z 466.868,A -85,B 0,C 180,E1 -12143.364,E2 -12143.364} C_VEL
LIN {X 0,Y 388.292,Z 455.011,A -85,B 0,C 180,E1 -12143.955,E2 -12143.955} C_VEL
LIN {X 0,Y 388.763,Z 444.763,A -85,B 0,C 180,E1 -12144.317,E2 -12144.317} C_VEL
LIN {X 0,Y 389.049,Z 428.08,A -85,B 0,C 180,E1 -12144.683,E2 -12144.683} C_VEL
LIN {X 0,Y 389.951,Z 370.707,A -85,B 0,C 180,E1 -12145.756,E2 -12145.756} C_VEL
LIN {X 0,Y 389.64,Z 366.844,A -85,B 0,C 180,E1 -12145.848,E2 -12145.848} C_VEL
LIN {X 0,Y 388.703,Z 363.108,A -85,B 0,C 180,E1 -12145.969,E2 -12145.969} C_VEL
LIN {X 0,Y 385.705,Z 356.006,A -85,B 0,C 180,E1 -12146.263,E2 -12146.263} C_VEL
LIN {X 0,Y 380.796,Z 345.343,A -85,B 0,C 180,E1 -12146.732,E2 -12146.732} C_VEL
LIN {X 0,Y 379.739,Z 341.554,A -85,B 0,C 180,E1 -12146.864,E2 -12146.864} C_VEL
LIN {X 0,Y 378.533,Z 335.359,A -85,B 0,C 180,E1 -12147.088,E2 -12147.088} C_VEL
LIN {X 0,Y 378.828,Z 330.929,A -85,B 0,C 180,E1 -12148.14,E2 -12148.14} C_VEL
LIN {X 0,Y 377.525,Z 322.025,A -85,B 0,C 180,E1 -12150.533,E2 -12150.533} C_VEL
LIN {X 0,Y 376.332,Z 316.134,A -85,B 0,C 180,E1 -12152.241,E2 -12152.241} C_VEL
LIN {X 0,Y 376.231,Z 316.116,A -85,B 0,C 180,E1 -12156.435,E2 -12156.435} C_VEL
LIN {X 0,Y 376.115,Z 316.137,A -85,B 0,C 180,E1 -12159.682,E2 -12159.682} C_VEL
LIN {X 0,Y 376.091,Z 316.139,A -85,B 0,C 180,E1 -12163.658,E2 -12163.658} C_VEL
LIN {X 0,Y 376.045,Z 316.143,A -85,B 0,C 180,E1 -12167.607,E2 -12167.607} C_VEL
LIN {X 0,Y 375.98,Z 316.15,A -85,B 0,C 180,E1 -12170.832,E2 -12170.832} C_VEL
LIN {X 0,Y 375.991,Z 316.144,A -85,B 0,C 180,E1 -12174.282,E2 -12174.282} C_VEL
LIN {X 0,Y 376.021,Z 316.147,A -85,B 0,C 180,E1 -12176.652,E2 -12176.652} C_VEL
LIN {X 0,Y 375.966,Z 316.148,A -85,B 0,C 180,E1 -12180.313,E2 -12180.313} C_VEL
LIN {X 0,Y 375.961,Z 316.139,A -85,B 0,C 180,E1 -12184.111,E2 -12184.111} C_VEL
LIN {X 0,Y 375.955,Z 316.15,A -85,B 0,C 180,E1 -12186.741,E2 -12186.741} C_VEL
LIN {X 0,Y 375.991,Z 316.143,A -85,B 0,C 180,E1 -12189.971,E2 -12189.971} C_VEL
LIN {X 0,Y 375.931,Z 316.148,A -85,B 0,C 180,E1 -12193.766,E2 -12193.766} C_VEL
LIN {X 0,Y 375.936,Z 316.155,A -85,B 0,C 180,E1 -12196.811,E2 -12196.811} C_VEL
LIN {X 0,Y 375.945,Z 316.135,A -85,B 0,C 180,E1 -12200.535,E2 -12200.535} C_VEL
LIN {X 0,Y 375.965,Z 316.152,A -85,B 0,C 180,E1 -12203.496,E2 -12203.496} C_VEL
LIN {X 0,Y 375.962,Z 316.15,A -85,B 0,C 180,E1 -12205.889,E2 -12205.889} C_VEL
LIN {X 0,Y 375.964,Z 316.131,A -85,B 0,C 180,E1 -12209.687,E2 -12209.687} C_VEL
LIN {X 0,Y 375.941,Z 316.144,A -85,B 0,C 180,E1 -12213.342,E2 -12213.342} C_VEL
LIN {X 0,Y 375.986,Z 316.146,A -85,B 0,C 180,E1 -12216.887,E2 -12216.887} C_VEL
LIN {X 0,Y 375.999,Z 316.131,A -85,B 0,C 180,E1 -12220.339,E2 -12220.339} C_VEL
LIN {X 0,Y 376.028,Z 316.129,A -85,B 0,C 180,E1 -12223.719,E2 -12223.719} C_VEL
LIN {X 0,Y 376.106,Z 316.133,A -85,B 0,C 180,E1 -12227.042,E2 -12227.042} C_VEL
LIN {X 0,Y 376.114,Z 316.123,A -85,B 0,C 180,E1 -12230.318,E2 -12230.318} C_VEL
LIN {X 0,Y 376.2,Z 316.096,A -85,B 0,C 180,E1 -12233.564,E2 -12233.564} C_VEL
LIN {X 0,Y 376.341,Z 316.1,A -85,B 0,C 180,E1 -12237.859,E2 -12237.859} C_VEL
LIN {X 0,Y 376.269,Z 316.107,A -85,B 0,C 180,E1 -12241.07,E2 -12241.07} C_VEL
LIN {X 0,Y 376.339,Z 316.099,A -85,B 0,C 180,E1 -12242.14,E2 -12242.14} C_VEL
LIN {X 0,Y 376.221,Z 316.101,A -85,B 0,C 180,E1 -12246.435,E2 -12246.435} C_VEL
LIN {X 0,Y 376.114,Z 316.133,A -85,B 0,C 180,E1 -12249.681,E2 -12249.681} C_VEL
LIN {X 0,Y 376.091,Z 316.122,A -85,B 0,C 180,E1 -12253.657,E2 -12253.657} C_VEL
LIN {X 0,Y 376.007,Z 316.139,A -85,B 0,C 180,E1 -12257.589,E2 -12257.589} C_VEL
LIN {X 0,Y 375.979,Z 316.146,A -85,B 0,C 180,E1 -12260.832,E2 -12260.832} C_VEL
LIN {X 0,Y 375.968,Z 316.136,A -85,B 0,C 180,E1 -12264.283,E2 -12264.283} C_VEL
LIN {X 0,Y 375.918,Z 316.155,A -85,B 0,C 180,E1 -12267.865,E2 -12267.865} C_VEL
LIN {X 0,Y 375.956,Z 316.144,A -85,B 0,C 180,E1 -12271.562,E2 -12271.562} C_VEL
LIN {X 0,Y 375.955,Z 316.155,A -85,B 0,C 180,E1 -12275.415,E2 -12275.415} C_VEL
LIN {X 0,Y 375.934,Z 316.153,A -85,B 0,C 180,E1 -12278.262,E2 -12278.262} C_VEL
LIN {X 0,Y 375.912,Z 316.158,A -85,B 0,C 180,E1 -12281.597,E2 -12281.597} C_VEL
LIN {X 0,Y 375.918,Z 316.158,A -85,B 0,C 180,E1 -12284.73,E2 -12284.73} C_VEL
LIN {X 0,Y 375.905,Z 316.158,A -85,B 0,C 180,E1 -12287.696,E2 -12287.696} C_VEL
LIN {X 0,Y 375.933,Z 316.158,A -85,B 0,C 180,E1 -12290.534,E2 -12290.534} C_VEL
LIN {X 0,Y 375.956,Z 316.153,A -85,B 0,C 180,E1 -12293.496,E2 -12293.496} C_VEL
LIN {X 0,Y 375.955,Z 316.147,A -85,B 0,C 180,E1 -12295.888,E2 -12295.888} C_VEL
LIN {X 0,Y 375.96,Z 316.151,A -85,B 0,C 180,E1 -12299.687,E2 -12299.687} C_VEL
LIN {X 0,Y 375.97,Z 316.301,A -85,B 0,C 180,E1 -12301.814,E2 -12301.814} C_VEL
LIN {X 0,Y 378.21,Z 327.189,A -85,B 0,C 180,E1 -12304.698,E2 -12304.698} C_VEL
LIN {X 0,Y 379.237,Z 333.257,A -85,B 0,C 180,E1 -12306.23,E2 -12306.23} C_VEL
LIN {X 0,Y 378.332,Z 344.948,A -85,B 0,C 180,E1 -12308.932,E2 -12308.932} C_VEL
LIN {X 0,Y 383.114,Z 373.789,A -85,B 0,C 180,E1 -12309.797,E2 -12309.797} C_VEL
LIN {X 0,Y 382.055,Z 447.931,A -85,B 0,C 180,E1 -12311.221,E2 -12311.221} C_VEL
LIN {X 0,Y 381.708,Z 460.531,A -85,B 0,C 180,E1 -12311.586,E2 -12311.586} C_VEL
LIN {X 0,Y 381.001,Z 471.798,A -85,B 0,C 180,E1 -12312.072,E2 -12312.072} C_VEL
LIN {X 0,Y 380.448,Z 481.936,A -85,B 0,C 180,E1 -12312.67,E2 -12312.67} C_VEL
LIN {X 0,Y 379.585,Z 492.477,A -85,B 0,C 180,E1 -12313.461,E2 -12313.461} C_VEL
LIN {X 0,Y 378.803,Z 502.375,A -85,B 0,C 180,E1 -12314.394,E2 -12314.394} C_VEL
LIN {X 0,Y 378.068,Z 510.52,A -85,B 0,C 180,E1 -12315.314,E2 -12315.314} C_VEL
LIN {X 0,Y 377.266,Z 519.439,A -85,B 0,C 180,E1 -12316.534,E2 -12316.534} C_VEL
LIN {X 0,Y 376.63,Z 526.107,A -85,B 0,C 180,E1 -12317.608,E2 -12317.608} C_VEL
LIN {X 0,Y 375.908,Z 533.087,A -85,B 0,C 180,E1 -12318.952,E2 -12318.952} C_VEL
LIN {X 0,Y 375.416,Z 538.921,A -85,B 0,C 180,E1 -12320.3,E2 -12320.3} C_VEL
LIN {X 0,Y 374.971,Z 544.579,A -85,B 0,C 180,E1 -12321.919,E2 -12321.919} C_VEL
LIN {X 0,Y 374.624,Z 549.742,A -85,B 0,C 180,E1 -12323.869,E2 -12323.869} C_VEL
LIN {X 0,Y 374.524,Z 553.222,A -85,B 0,C 180,E1 -12325.695,E2 -12325.695} C_VEL
LIN {X 0,Y 374.429,Z 554.789,A -85,B 0,C 180,E1 -12326.772,E2 -12326.772} C_VEL
LIN {X 0,Y 374.447,Z 556.415,A -85,B 0,C 180,E1 -12328.924,E2 -12328.924} C_VEL
LIN {X 0,Y 374.468,Z 556.732,A -85,B 0,C 180,E1 -12330,E2 -12330} C_VEL
LIN {X 0,Y 374.408,Z 555.987,A -85,B 0,C 180,E1 -12332.151,E2 -12332.151} C_VEL
LIN {X 0,Y 374.43,Z 555.013,A -85,B 0,C 180,E1 -12333.228,E2 -12333.228} C_VEL
LIN {X 0,Y 374.603,Z 551.895,A -85,B 0,C 180,E1 -12335.383,E2 -12335.383} C_VEL
LIN {X 0,Y 374.768,Z 548.356,A -85,B 0,C 180,E1 -12337.001,E2 -12337.001} C_VEL
LIN {X 0,Y 375.126,Z 543.713,A -85,B 0,C 180,E1 -12338.62,E2 -12338.62} C_VEL
LIN {X 0,Y 375.656,Z 537.814,A -85,B 0,C 180,E1 -12340.238,E2 -12340.238} C_VEL
LIN {X 0,Y 376.346,Z 530.432,A -85,B 0,C 180,E1 -12341.854,E2 -12341.854} C_VEL
LIN {X 0,Y 377.183,Z 522.962,A -85,B 0,C 180,E1 -12343.194,E2 -12343.194} C_VEL
LIN {X 0,Y 378.013,Z 514.691,A -85,B 0,C 180,E1 -12344.429,E2 -12344.429} C_VEL
LIN {X 0,Y 378.848,Z 506.37,A -85,B 0,C 180,E1 -12345.466,E2 -12345.466} C_VEL
LIN {X 0,Y 379.653,Z 497.428,A -85,B 0,C 180,E1 -12346.398,E2 -12346.398} C_VEL
LIN {X 0,Y 380.519,Z 488.182,A -85,B 0,C 180,E1 -12347.188,E2 -12347.188} C_VEL
LIN {X 0,Y 381.408,Z 476.346,A -85,B 0,C 180,E1 -12347.977,E2 -12347.977} C_VEL
LIN {X 0,Y 382.087,Z 465.232,A -85,B 0,C 180,E1 -12348.534,E2 -12348.534} C_VEL
LIN {X 0,Y 382.58,Z 455.412,A -85,B 0,C 180,E1 -12348.891,E2 -12348.891} C_VEL
LIN {X 0,Y 382.978,Z 437.637,A -85,B 0,C 180,E1 -12349.288,E2 -12349.288} C_VEL
LIN {X 0,Y 383.826,Z 373.111,A -85,B 0,C 180,E1 -12350.541,E2 -12350.541} C_VEL
LIN {X 0,Y 379.265,Z 347.721,A -85,B 0,C 180,E1 -12351.342,E2 -12351.342} C_VEL
LIN {X 0,Y 378.687,Z 344.483,A -85,B 0,C 180,E1 -12351.494,E2 -12351.494} C_VEL
LIN {X 0,Y 379.507,Z 334.368,A -85,B 0,C 180,E1 -12353.752,E2 -12353.752} C_VEL
LIN {X 0,Y 378.018,Z 325.76,A -85,B 0,C 180,E1 -12355.907,E2 -12355.907} C_VEL
LIN {X 0,Y 375.976,Z 316.308,A -85,B 0,C 180,E1 -12358.417,E2 -12358.417} C_VEL
LIN {X 0,Y 375.955,Z 316.152,A -85,B 0,C 180,E1 -12361.562,E2 -12361.562} C_VEL
LIN {X 0,Y 375.955,Z 316.154,A -85,B 0,C 180,E1 -12365.416,E2 -12365.416} C_VEL
LIN {X 0,Y 375.971,Z 316.152,A -85,B 0,C 180,E1 -12368.27,E2 -12368.27} C_VEL
LIN {X 0,Y 375.922,Z 316.159,A -85,B 0,C 180,E1 -12371.599,E2 -12371.599} C_VEL
